LIN {X 0,Y 318.182,Z 547.875,A -85,B 0,C 180,E1 -15955.427,E2 -15955.427} C_VEL
LIN {X 0,Y 320.026,Z 530.036,A -85,B 0,C 180,E1 -15956.582,E2 -15956.582} C_VEL
LIN {X 0,Y 321.174,Z 516.208,A -85,B 0,C 180,E1 -15957.226,E2 -15957.226} C_VEL
LIN {X 0,Y 322.105,Z 502.779,A -85,B 0,C 180,E1 -15957.713,E2 -15957.713} C_VEL
LIN {X 0,Y 330.031,Z 435.019,A -85,B 0,C 180,E1 -15960.427,E2 -15960.427} C_VEL
LIN {X 0,Y 332.161,Z 417.671,A -85,B 0,C 180,E1 -15961.143,E2 -15961.143} C_VEL
LIN {X 0,Y 332.144,Z 415.549,A -85,B 0,C 180,E1 -15961.342,E2 -15961.342} C_VEL
LIN {X 0,Y 332.385,Z 414.109,A -85,B 0,C 180,E1 -15961.515,E2 -15961.515} C_VEL
LIN {X 0,Y 332.046,Z 411.059,A -85,B 0,C 180,E1 -15962.153,E2 -15962.153} C_VEL
LIN {X 0,Y 331.408,Z 405.664,A -85,B 0,C 180,E1 -15963.462,E2 -15963.462} C_VEL
LIN {X 0,Y 330.123,Z 402.878,A -85,B 0,C 180,E1 -15964.617,E2 -15964.617} C_VEL
LIN {X 0,Y 327.789,Z 399.05,A -85,B 0,C 180,E1 -15966.896,E2 -15966.896} C_VEL
LIN {X 0,Y 326.226,Z 396.525,A -85,B 0,C 180,E1 -15969.144,E2 -15969.144} C_VEL
LIN {X 0,Y 325.461,Z 395.342,A -85,B 0,C 180,E1 -15970.906,E2 -15970.906} C_VEL
LIN {X 0,Y 324.942,Z 395.007,A -85,B 0,C 180,E1 -15972.662,E2 -15972.662} C_VEL
LIN {X 0,Y 324.638,Z 395.462,A -85,B 0,C 180,E1 -15974.405,E2 -15974.405} C_VEL
LIN {X 0,Y 324.653,Z 396.483,A -85,B 0,C 180,E1 -15976.154,E2 -15976.154} C_VEL
LIN {X 0,Y 324.963,Z 398.076,A -85,B 0,C 180,E1 -15977.899,E2 -15977.899} C_VEL
LIN {X 0,Y 325.669,Z 401.15,A -85,B 0,C 180,E1 -15980.222,E2 -15980.222} C_VEL
LIN {X 0,Y 326.682,Z 406.362,A -85,B 0,C 180,E1 -15982.96,E2 -15982.96} C_VEL
LIN {X 0,Y 327.403,Z 411.448,A -85,B 0,C 180,E1 -15985.029,E2 -15985.029} C_VEL
LIN {X 0,Y 327.833,Z 416.51,A -85,B 0,C 180,E1 -15986.73,E2 -15986.73} C_VEL
LIN {X 0,Y 327.465,Z 419.21,A -85,B 0,C 180,E1 -15987.399,E2 -15987.399} C_VEL
LIN {X 0,Y 329.647,Z 433.874,A -85,B 0,C 180,E1 -15989.149,E2 -15989.149} C_VEL
LIN {X 0,Y 331.611,Z 449.295,A -85,B 0,C 180,E1 -15990.644,E2 -15990.644} C_VEL
LIN {X 0,Y 332.453,Z 459.55,A -85,B 0,C 180,E1 -15991.459,E2 -15991.459} C_VEL
LIN {X 0,Y 324.883,Z 534.704,A -85,B 0,C 180,E1 -15994.364,E2 -15994.364} C_VEL
LIN {X 0,Y 322.805,Z 549.723,A -85,B 0,C 180,E1 -15995.222,E2 -15995.222} C_VEL
LIN {X 0,Y 320.608,Z 562.727,A -85,B 0,C 180,E1 -15996.247,E2 -15996.247} C_VEL
LIN {X 0,Y 318.379,Z 574.516,A -85,B 0,C 180,E1 -15997.447,E2 -15997.447} C_VEL
LIN {X 0,Y 315.803,Z 586.406,A -85,B 0,C 180,E1 -15998.97,E2 -15998.97} C_VEL
LIN {X 0,Y 313.366,Z 596.431,A -85,B 0,C 180,E1 -16000.571,E2 -16000.571} C_VEL
LIN {X 0,Y 311.237,Z 604.933,A -85,B 0,C 180,E1 -16002.251,E2 -16002.251} C_VEL
LIN {X 0,Y 309.091,Z 612.857,A -85,B 0,C 180,E1 -16004.166,E2 -16004.166} C_VEL
LIN {X 0,Y 307.572,Z 619.204,A -85,B 0,C 180,E1 -16006.118,E2 -16006.118} C_VEL
LIN {X 0,Y 306.235,Z 624.295,A -85,B 0,C 180,E1 -16008.08,E2 -16008.08} C_VEL
LIN {X 0,Y 305.158,Z 628.243,A -85,B 0,C 180,E1 -16010.054,E2 -16010.054} C_VEL
LIN {X 0,Y 304.385,Z 631.13,A -85,B 0,C 180,E1 -16012.037,E2 -16012.037} C_VEL
LIN {X 0,Y 303.995,Z 632.859,A -85,B 0,C 180,E1 -16013.787,E2 -16013.787} C_VEL
LIN {X 0,Y 303.692,Z 633.934,A -85,B 0,C 180,E1 -16016.019,E2 -16016.019} C_VEL
LIN {X 0,Y 303.606,Z 633.986,A -85,B 0,C 180,E1 -16017.347,E2 -16017.347} C_VEL
LIN {X 0,Y 303.535,Z 633.619,A -85,B 0,C 180,E1 -16018.673,E2 -16018.673} C_VEL
LIN {X 0,Y 303.515,Z 632.811,A -85,B 0,C 180,E1 -16020,E2 -16020} C_VEL
LIN {X 0,Y 303.532,Z 631.523,A -85,B 0,C 180,E1 -16021.327,E2 -16021.327} C_VEL
LIN {X 0,Y 303.667,Z 628.745,A -85,B 0,C 180,E1 -16023.317,E2 -16023.317} C_VEL
LIN {X 0,Y 303.691,Z 624.826,A -85,B 0,C 180,E1 -16025.311,E2 -16025.311} C_VEL
LIN {X 0,Y 303.942,Z 619.686,A -85,B 0,C 180,E1 -16027.307,E2 -16027.307} C_VEL
LIN {X 0,Y 304.298,Z 613.15,A -85,B 0,C 180,E1 -16029.304,E2 -16029.304} C_VEL
LIN {X 0,Y 304.814,Z 604.894,A -85,B 0,C 180,E1 -16031.302,E2 -16031.302} C_VEL
LIN {X 0,Y 305.528,Z 596.499,A -85,B 0,C 180,E1 -16032.961,E2 -16032.961} C_VEL
LIN {X 0,Y 306.26,Z 587.38,A -85,B 0,C 180,E1 -16034.451,E2 -16034.451} C_VEL
LIN {X 0,Y 307.145,Z 576.203,A -85,B 0,C 180,E1 -16035.937,E2 -16035.937} C_VEL
LIN {X 0,Y 308.041,Z 563.777,A -85,B 0,C 180,E1 -16037.253,E2 -16037.253} C_VEL
LIN {X 0,Y 308.857,Z 550.689,A -85,B 0,C 180,E1 -16038.319,E2 -16038.319} C_VEL
LIN {X 0,Y 309.631,Z 537.051,A -85,B 0,C 180,E1 -16039.129,E2 -16039.129} C_VEL
LIN {X 0,Y 310.165,Z 522.846,A -85,B 0,C 180,E1 -16039.697,E2 -16039.697} C_VEL
LIN {X 0,Y 312.404,Z 451.025,A -85,B 0,C 180,E1 -16042.076,E2 -16042.076} C_VEL
LIN {X 0,Y 309.46,Z 422.574,A -85,B 0,C 180,E1 -16043.175,E2 -16043.175} C_VEL
LIN {X 0,Y 309.339,Z 419.877,A -85,B 0,C 180,E1 -16043.339,E2 -16043.339} C_VEL
LIN {X 0,Y 310.896,Z 400.877,A -85,B 0,C 180,E1 -16046.879,E2 -16046.879} C_VEL
LIN {X 0,Y 311.786,Z 389.598,A -85,B 0,C 180,E1 -16048.988,E2 -16048.988} C_VEL
LIN {X 0,Y 308.814,Z 375.793,A -85,B 0,C 180,E1 -16051.827,E2 -16051.827} C_VEL
LIN {X 0,Y 305.536,Z 361.201,A -85,B 0,C 180,E1 -16054.969,E2 -16054.969} C_VEL
LIN {X 0,Y 305.455,Z 361.063,A -85,B 0,C 180,E1 -16058.528,E2 -16058.528} C_VEL
LIN {X 0,Y 305.461,Z 361.055,A -85,B 0,C 180,E1 -16062.585,E2 -16062.585} C_VEL
LIN {X 0,Y 305.431,Z 361.045,A -85,B 0,C 180,E1 -16066.344,E2 -16066.344} C_VEL
LIN {X 0,Y 305.464,Z 361.04,A -85,B 0,C 180,E1 -16069.892,E2 -16069.892} C_VEL
LIN {X 0,Y 305.509,Z 361.129,A -85,B 0,C 180,E1 -16073.831,E2 -16073.831} C_VEL
LIN {X 0,Y 306.963,Z 366.882,A -85,B 0,C 180,E1 -16075.879,E2 -16075.879} C_VEL
LIN {X 0,Y 308.34,Z 372.284,A -85,B 0,C 180,E1 -16077.59,E2 -16077.59} C_VEL
LIN {X 0,Y 316.163,Z 388.914,A -85,B 0,C 180,E1 -16078.96,E2 -16078.96} C_VEL
LIN {X 0,Y 322.479,Z 404.145,A -85,B 0,C 180,E1 -16080.018,E2 -16080.018} C_VEL
LIN {X 0,Y 324.452,Z 415.875,A -85,B 0,C 180,E1 -16080.511,E2 -16080.511} C_VEL
LIN {X 0,Y 321.971,Z 498.445,A -85,B 0,C 180,E1 -16082.319,E2 -16082.319} C_VEL
LIN {X 0,Y 321.342,Z 514.068,A -85,B 0,C 180,E1 -16082.746,E2 -16082.746} C_VEL
LIN {X 0,Y 320.191,Z 527.937,A -85,B 0,C 180,E1 -16083.345,E2 -16083.345} C_VEL
LIN {X 0,Y 318.78,Z 541.464,A -85,B 0,C 180,E1 -16084.187,E2 -16084.187} C_VEL
LIN {X 0,Y 317.108,Z 554.588,A -85,B 0,C 180,E1 -16085.277,E2 -16085.277} C_VEL
LIN {X 0,Y 315.332,Z 566.41,A -85,B 0,C 180,E1 -16086.521,E2 -16086.521} C_VEL
LIN {X 0,Y 313.251,Z 578.455,A -85,B 0,C 180,E1 -16088.098,E2 -16088.098} C_VEL
LIN {X 0,Y 311.184,Z 589.311,A -85,B 0,C 180,E1 -16089.852,E2 -16089.852} C_VEL
LIN {X 0,Y 309.222,Z 599.086,A -85,B 0,C 180,E1 -16091.788,E2 -16091.788} C_VEL
LIN {X 0,Y 307.761,Z 606.494,A -85,B 0,C 180,E1 -16093.559,E2 -16093.559} C_VEL
LIN {X 0,Y 306.497,Z 613.955,A -85,B 0,C 180,E1 -16095.728,E2 -16095.728} C_VEL
LIN {X 0,Y 305.183,Z 620.391,A -85,B 0,C 180,E1 -16098.037,E2 -16098.037} C_VEL
LIN {X 0,Y 304.31,Z 626.095,A -85,B 0,C 180,E1 -16100.695,E2 -16100.695} C_VEL
LIN {X 0,Y 303.832,Z 630.239,A -85,B 0,C 180,E1 -16103.357,E2 -16103.357} C_VEL
LIN {X 0,Y 303.606,Z 632.954,A -85,B 0,C 180,E1 -16106.016,E2 -16106.016} C_VEL
LIN {X 0,Y 303.527,Z 634.316,A -85,B 0,C 180,E1 -16108.672,E2 -16108.672} C_VEL
LIN {X 0,Y 303.526,Z 634.349,A -85,B 0,C 180,E1 -16111.325,E2 -16111.325} C_VEL
LIN {X 0,Y 303.603,Z 633.053,A -85,B 0,C 180,E1 -16113.98,E2 -16113.98} C_VEL
LIN {X 0,Y 303.83,Z 630.396,A -85,B 0,C 180,E1 -16116.64,E2 -16116.64} C_VEL
LIN {X 0,Y 304.303,Z 626.307,A -85,B 0,C 180,E1 -16119.302,E2 -16119.302} C_VEL
LIN {X 0,Y 305.143,Z 620.663,A -85,B 0,C 180,E1 -16121.962,E2 -16121.962} C_VEL
LIN {X 0,Y 306.457,Z 614.298,A -85,B 0,C 180,E1 -16124.27,E2 -16124.27} C_VEL
LIN {X 0,Y 307.777,Z 606.859,A -85,B 0,C 180,E1 -16126.451,E2 -16126.451} C_VEL
LIN {X 0,Y 309.476,Z 598.103,A -85,B 0,C 180,E1 -16128.536,E2 -16128.536} C_VEL
LIN {X 0,Y 311.411,Z 588.131,A -85,B 0,C 180,E1 -16130.474,E2 -16130.474} C_VEL
LIN {X 0,Y 313.545,Z 577.03,A -85,B 0,C 180,E1 -16132.223,E2 -16132.223} C_VEL
LIN {X 0,Y 315.477,Z 565.984,A -85,B 0,C 180,E1 -16133.638,E2 -16133.638} C_VEL
LIN {X 0,Y 317.275,Z 553.988,A -85,B 0,C 180,E1 -16134.888,E2 -16134.888} C_VEL
LIN {X 0,Y 318.927,Z 540.711,A -85,B 0,C 180,E1 -16135.973,E2 -16135.973} C_VEL
LIN {X 0,Y 320.323,Z 526.914,A -85,B 0,C 180,E1 -16136.815,E2 -16136.815} C_VEL
LIN {X 0,Y 321.461,Z 512.549,A -85,B 0,C 180,E1 -16137.416,E2 -16137.416} C_VEL
LIN {X 0,Y 322.286,Z 492.491,A -85,B 0,C 180,E1 -16137.913,E2 -16137.913} C_VEL
LIN {X 0,Y 322.395,Z 488.057,A -85,B 0,C 180,E1 -16138.012,E2 -16138.012} C_VEL
LIN {X 0,Y 322.01,Z 482.254,A -85,B 0,C 180,E1 -16138.192,E2 -16138.192} C_VEL
LIN {X 0,Y 317.564,Z 463.594,A -85,B 0,C 180,E1 -16139.095,E2 -16139.095} C_VEL
LIN {X 0,Y 317.105,Z 457.794,A -85,B 0,C 180,E1 -16139.288,E2 -16139.288} C_VEL
LIN {X 0,Y 318.252,Z 415.603,A -85,B 0,C 180,E1 -16140.246,E2 -16140.246} C_VEL
LIN {X 0,Y 316.291,Z 405.8,A -85,B 0,C 180,E1 -16140.706,E2 -16140.706} C_VEL
LIN {X 0,Y 309.273,Z 389.276,A -85,B 0,C 180,E1 -16141.923,E2 -16141.923} C_VEL
LIN {X 0,Y 301.176,Z 372.441,A -85,B 0,C 180,E1 -16143.389,E2 -16143.389} C_VEL
LIN {X 0,Y 300.133,Z 368.625,A -85,B 0,C 180,E1 -16144.591,E2 -16144.591} C_VEL
LIN {X 0,Y 298.468,Z 361.978,A -85,B 0,C 180,E1 -16147.021,E2 -16147.021} C_VEL
LIN {X 0,Y 298.451,Z 361.921,A -85,B 0,C 180,E1 -16151.248,E2 -16151.248} C_VEL
LIN {X 0,Y 298.483,Z 361.897,A -85,B 0,C 180,E1 -16155.059,E2 -16155.059} C_VEL
LIN {X 0,Y 298.452,Z 361.934,A -85,B 0,C 180,E1 -16158.895,E2 -16158.895} C_VEL
LIN {X 0,Y 298.458,Z 361.893,A -85,B 0,C 180,E1 -16163.186,E2 -16163.186} C_VEL
LIN {X 0,Y 298.388,Z 361.939,A -85,B 0,C 180,E1 -16167.199,E2 -16167.199} C_VEL
LIN {X 0,Y 298.423,Z 361.878,A -85,B 0,C 180,E1 -16170.614,E2 -16170.614} C_VEL
LIN {X 0,Y 298.475,Z 361.904,A -85,B 0,C 180,E1 -16173.473,E2 -16173.473} C_VEL
LIN {X 0,Y 298.427,Z 361.936,A -85,B 0,C 180,E1 -16176.696,E2 -16176.696} C_VEL
LIN {X 0,Y 298.53,Z 361.919,A -85,B 0,C 180,E1 -16180.756,E2 -16180.756} C_VEL
LIN {X 0,Y 298.583,Z 361.897,A -85,B 0,C 180,E1 -16184.994,E2 -16184.994} C_VEL
LIN {X 0,Y 298.585,Z 361.902,A -85,B 0,C 180,E1 -16189.146,E2 -16189.146} C_VEL
LIN {X 0,Y 298.748,Z 361.884,A -85,B 0,C 180,E1 -16191.886,E2 -16191.886} C_VEL
LIN {X 0,Y 298.652,Z 361.905,A -85,B 0,C 180,E1 -16194.599,E2 -16194.599} C_VEL
LIN {X 0,Y 298.917,Z 361.868,A -85,B 0,C 180,E1 -16198.653,E2 -16198.653} C_VEL
LIN {X 0,Y 299.034,Z 361.86,A -85,B 0,C 180,E1 -16200,E2 -16200} C_VEL
LIN {X 0,Y 298.828,Z 361.868,A -85,B 0,C 180,E1 -16202.696,E2 -16202.696} C_VEL
LIN {X 0,Y 298.788,Z 361.891,A -85,B 0,C 180,E1 -16206.754,E2 -16206.754} C_VEL
LIN {X 0,Y 298.67,Z 361.883,A -85,B 0,C 180,E1 -16209.481,E2 -16209.481} C_VEL
LIN {X 0,Y 298.543,Z 361.914,A -85,B 0,C 180,E1 -16213.616,E2 -16213.616} C_VEL
LIN {X 0,Y 298.538,Z 361.903,A -85,B 0,C 180,E1 -16216.409,E2 -16216.409} C_VEL
LIN {X 0,Y 298.502,Z 361.92,A -85,B 0,C 180,E1 -16219.656,E2 -16219.656} C_VEL
LIN {X 0,Y 298.448,Z 361.932,A -85,B 0,C 180,E1 -16223.598,E2 -16223.598} C_VEL
LIN {X 0,Y 298.473,Z 361.904,A -85,B 0,C 180,E1 -16226.576,E2 -16226.576} C_VEL
LIN {X 0,Y 298.394,Z 361.882,A -85,B 0,C 180,E1 -16229.644,E2 -16229.644} C_VEL
LIN {X 0,Y 298.384,Z 361.938,A -85,B 0,C 180,E1 -16232.802,E2 -16232.802} C_VEL
LIN {X 0,Y 298.457,Z 361.893,A -85,B 0,C 180,E1 -16236.814,E2 -16236.814} C_VEL
LIN {X 0,Y 298.452,Z 361.934,A -85,B 0,C 180,E1 -16241.25,E2 -16241.25} C_VEL
LIN {X 0,Y 298.482,Z 361.897,A -85,B 0,C 180,E1 -16245.062,E2 -16245.062} C_VEL
LIN {X 0,Y 298.45,Z 361.92,A -85,B 0,C 180,E1 -16248.898,E2 -16248.898} C_VEL
LIN {X 0,Y 298.468,Z 362.013,A -85,B 0,C 180,E1 -16253.044,E2 -16253.044} C_VEL
LIN {X 0,Y 300.449,Z 369.766,A -85,B 0,C 180,E1 -16255.85,E2 -16255.85} C_VEL
LIN {X 0,Y 301.11,Z 372.24,A -85,B 0,C 180,E1 -16256.627,E2 -16256.627} C_VEL
LIN {X 0,Y 308.478,Z 387.538,A -85,B 0,C 180,E1 -16257.984,E2 -16257.984} C_VEL
LIN {X 0,Y 316.033,Z 405.034,A -85,B 0,C 180,E1 -16259.291,E2 -16259.291} C_VEL
LIN {X 0,Y 317.506,Z 411.383,A -85,B 0,C 180,E1 -16259.612,E2 -16259.612} C_VEL
LIN {X 0,Y 318.332,Z 416.622,A -85,B 0,C 180,E1 -16259.833,E2 -16259.833} C_VEL
LIN {X 0,Y 315.898,Z 494.268,A -85,B 0,C 180,E1 -16261.562,E2 -16261.562} C_VEL
LIN {X 0,Y 315.218,Z 512.539,A -85,B 0,C 180,E1 -16262.039,E2 -16262.039} C_VEL
LIN {X 0,Y 314.041,Z 526.906,A -85,B 0,C 180,E1 -16262.649,E2 -16262.649} C_VEL
LIN {X 0,Y 312.551,Z 540.139,A -85,B 0,C 180,E1 -16263.457,E2 -16263.457} C_VEL
LIN {X 0,Y 310.881,Z 553.549,A -85,B 0,C 180,E1 -16264.565,E2 -16264.565} C_VEL
LIN {X 0,Y 309.072,Z 565.636,A -85,B 0,C 180,E1 -16265.841,E2 -16265.841} C_VEL
LIN {X 0,Y 306.791,Z 577.83,A -85,B 0,C 180,E1 -16267.438,E2 -16267.438} C_VEL
LIN {X 0,Y 304.814,Z 587.901,A -85,B 0,C 180,E1 -16269.063,E2 -16269.063} C_VEL
LIN {X 0,Y 302.738,Z 597.911,A -85,B 0,C 180,E1 -16271.036,E2 -16271.036} C_VEL
LIN {X 0,Y 300.823,Z 607.229,A -85,B 0,C 180,E1 -16273.308,E2 -16273.308} C_VEL
LIN {X 0,Y 299.357,Z 615.173,A -85,B 0,C 180,E1 -16275.731,E2 -16275.731} C_VEL
LIN {X 0,Y 298.172,Z 620.557,A -85,B 0,C 180,E1 -16277.755,E2 -16277.755} C_VEL
LIN {X 0,Y 297.268,Z 626.225,A -85,B 0,C 180,E1 -16280.476,E2 -16280.476} C_VEL
LIN {X 0,Y 296.745,Z 630.336,A -85,B 0,C 180,E1 -16283.201,E2 -16283.201} C_VEL
LIN {X 0,Y 296.511,Z 633.016,A -85,B 0,C 180,E1 -16285.924,E2 -16285.924} C_VEL
LIN {X 0,Y 296.447,Z 634.338,A -85,B 0,C 180,E1 -16288.643,E2 -16288.643} C_VEL
LIN {X 0,Y 296.448,Z 634.33,A -85,B 0,C 180,E1 -16291.36,E2 -16291.36} C_VEL
LIN {X 0,Y 296.625,Z 632.445,A -85,B 0,C 180,E1 -16295.666,E2 -16295.666} C_VEL
LIN {X 0,Y 296.843,Z 631.726,A -85,B 0,C 180,E1 -16296.8,E2 -16296.8} C_VEL
LIN {X 0,Y 297.059,Z 630.455,A -85,B 0,C 180,E1 -16298.162,E2 -16298.162} C_VEL
LIN {X 0,Y 297.678,Z 627.768,A -85,B 0,C 180,E1 -16300.201,E2 -16300.201} C_VEL
LIN {X 0,Y 298.488,Z 624.041,A -85,B 0,C 180,E1 -16302.236,E2 -16302.236} C_VEL
LIN {X 0,Y 299.721,Z 619.19,A -85,B 0,C 180,E1 -16304.255,E2 -16304.255} C_VEL
LIN {X 0,Y 301.314,Z 612.169,A -85,B 0,C 180,E1 -16306.556,E2 -16306.556} C_VEL
LIN {X 0,Y 303.075,Z 604.298,A -85,B 0,C 180,E1 -16308.595,E2 -16308.595} C_VEL
LIN {X 0,Y 305.146,Z 594.851,A -85,B 0,C 180,E1 -16310.564,E2 -16310.564} C_VEL
LIN {X 0,Y 307.109,Z 585.333,A -85,B 0,C 180,E1 -16312.186,E2 -16312.186} C_VEL
LIN {X 0,Y 309.295,Z 573.702,A -85,B 0,C 180,E1 -16313.788,E2 -16313.788} C_VEL
LIN {X 0,Y 311.179,Z 561.561,A -85,B 0,C 180,E1 -16315.16,E2 -16315.16} C_VEL
LIN {X 0,Y 312.961,Z 548.604,A -85,B 0,C 180,E1 -16316.294,E2 -16316.294} C_VEL
LIN {X 0,Y 314.492,Z 534.098,A -85,B 0,C 180,E1 -16317.267,E2 -16317.267} C_VEL
LIN {X 0,Y 316.409,Z 512.855,A -85,B 0,C 180,E1 -16318.256,E2 -16318.256} C_VEL
LIN {X 0,Y 328.061,Z 420.09,A -85,B 0,C 180,E1 -16322.059,E2 -16322.059} C_VEL
LIN {X 0,Y 327.883,Z 417.132,A -85,B 0,C 180,E1 -16322.362,E2 -16322.362} C_VEL
LIN {X 0,Y 327.312,Z 413.657,A -85,B 0,C 180,E1 -16323.133,E2 -16323.133} C_VEL
LIN {X 0,Y 326.869,Z 410.419,A -85,B 0,C 180,E1 -16323.99,E2 -16323.99} C_VEL
LIN {X 0,Y 324.961,Z 406.805,A -85,B 0,C 180,E1 -16325.729,E2 -16325.729} C_VEL
LIN {X 0,Y 322.672,Z 403.199,A -85,B 0,C 180,E1 -16328.362,E2 -16328.362} C_VEL
LIN {X 0,Y 321.345,Z 401.123,A -85,B 0,C 180,E1 -16331.006,E2 -16331.006} C_VEL
LIN {X 0,Y 320.772,Z 400.777,A -85,B 0,C 180,E1 -16332.783,E2 -16332.783} C_VEL
LIN {X 0,Y 320.308,Z 401.68,A -85,B 0,C 180,E1 -16335.402,E2 -16335.402} C_VEL
LIN {X 0,Y 320.558,Z 404.041,A -85,B 0,C 180,E1 -16338.197,E2 -16338.197} C_VEL
LIN {X 0,Y 321.17,Z 407.324,A -85,B 0,C 180,E1 -16340.61,E2 -16340.61} C_VEL
LIN {X 0,Y 321.833,Z 411.838,A -85,B 0,C 180,E1 -16342.963,E2 -16342.963} C_VEL
LIN {X 0,Y 322.325,Z 416.005,A -85,B 0,C 180,E1 -16344.7,E2 -16344.7} C_VEL
LIN {X 0,Y 322.667,Z 419.697,A -85,B 0,C 180,E1 -16345.94,E2 -16345.94} C_VEL
LIN {X 0,Y 323.66,Z 423.168,A -85,B 0,C 180,E1 -16346.604,E2 -16346.604} C_VEL
LIN {X 0,Y 325.648,Z 437.927,A -85,B 0,C 180,E1 -16348.394,E2 -16348.394} C_VEL
LIN {X 0,Y 327.174,Z 452.09,A -85,B 0,C 180,E1 -16349.814,E2 -16349.814} C_VEL
LIN {X 0,Y 327.787,Z 460.947,A -85,B 0,C 180,E1 -16350.55,E2 -16350.55} C_VEL
LIN {X 0,Y 319.743,Z 534.694,A -85,B 0,C 180,E1 -16353.482,E2 -16353.482} C_VEL
LIN {X 0,Y 317.564,Z 549.543,A -85,B 0,C 180,E1 -16354.346,E2 -16354.346} C_VEL
LIN {X 0,Y 315.066,Z 563.279,A -85,B 0,C 180,E1 -16355.452,E2 -16355.452} C_VEL
LIN {X 0,Y 312.672,Z 574.881,A -85,B 0,C 180,E1 -16356.662,E2 -16356.662} C_VEL
LIN {X 0,Y 309.938,Z 586.634,A -85,B 0,C 180,E1 -16358.204,E2 -16358.204} C_VEL
LIN {X 0,Y 307.202,Z 597.114,A -85,B 0,C 180,E1 -16359.93,E2 -16359.93} C_VEL
LIN {X 0,Y 304.647,Z 606.45,A -85,B 0,C 180,E1 -16361.854,E2 -16361.854} C_VEL
LIN {X 0,Y 302.36,Z 614.023,A -85,B 0,C 180,E1 -16363.804,E2 -16363.804} C_VEL
LIN {X 0,Y 300.743,Z 620.12,A -85,B 0,C 180,E1 -16365.796,E2 -16365.796} C_VEL
LIN {X 0,Y 299.343,Z 625,A -85,B 0,C 180,E1 -16367.801,E2 -16367.801} C_VEL
LIN {X 0,Y 298.188,Z 628.763,A -85,B 0,C 180,E1 -16369.819,E2 -16369.819} C_VEL
LIN {X 0,Y 297.374,Z 631.476,A -85,B 0,C 180,E1 -16371.848,E2 -16371.848} C_VEL
LIN {X 0,Y 296.88,Z 633.192,A -85,B 0,C 180,E1 -16373.869,E2 -16373.869} C_VEL
LIN {X 0,Y 296.598,Z 633.959,A -85,B 0,C 180,E1 -16375.924,E2 -16375.924} C_VEL
LIN {X 0,Y 296.514,Z 633.931,A -85,B 0,C 180,E1 -16377.283,E2 -16377.283} C_VEL
LIN {X 0,Y 296.457,Z 633.467,A -85,B 0,C 180,E1 -16378.642,E2 -16378.642} C_VEL
LIN {X 0,Y 296.434,Z 632.529,A -85,B 0,C 180,E1 -16380,E2 -16380} C_VEL
LIN {X 0,Y 296.454,Z 631.163,A -85,B 0,C 180,E1 -16381.359,E2 -16381.359} C_VEL
LIN {X 0,Y 296.602,Z 628.229,A -85,B 0,C 180,E1 -16383.396,E2 -16383.396} C_VEL
LIN {X 0,Y 296.672,Z 623.427,A -85,B 0,C 180,E1 -16385.744,E2 -16385.744} C_VEL
LIN {X 0,Y 296.937,Z 617.765,A -85,B 0,C 180,E1 -16387.822,E2 -16387.822} C_VEL
LIN {X 0,Y 297.319,Z 610.722,A -85,B 0,C 180,E1 -16389.868,E2 -16389.868} C_VEL
LIN {X 0,Y 297.826,Z 603.52,A -85,B 0,C 180,E1 -16391.571,E2 -16391.571} C_VEL
LIN {X 0,Y 298.566,Z 594.808,A -85,B 0,C 180,E1 -16393.268,E2 -16393.268} C_VEL
LIN {X 0,Y 299.482,Z 584.188,A -85,B 0,C 180,E1 -16394.96,E2 -16394.96} C_VEL
LIN {X 0,Y 300.336,Z 572.527,A -85,B 0,C 180,E1 -16396.45,E2 -16396.45} C_VEL
LIN {X 0,Y 301.219,Z 560.631,A -85,B 0,C 180,E1 -16397.657,E2 -16397.657} C_VEL
LIN {X 0,Y 302.001,Z 547.74,A -85,B 0,C 180,E1 -16398.662,E2 -16398.662} C_VEL
LIN {X 0,Y 302.784,Z 533.872,A -85,B 0,C 180,E1 -16399.447,E2 -16399.447} C_VEL
LIN {X 0,Y 303.969,Z 496.409,A -85,B 0,C 180,E1 -16400.779,E2 -16400.779} C_VEL
LIN {X 0,Y 305.461,Z 451.797,A -85,B 0,C 180,E1 -16402.315,E2 -16402.315} C_VEL
LIN {X 0,Y 302.673,Z 424.414,A -85,B 0,C 180,E1 -16403.408,E2 -16403.408} C_VEL
LIN {X 0,Y 302.372,Z 419.92,A -85,B 0,C 180,E1 -16403.637,E2 -16403.637} C_VEL
LIN {X 0,Y 303.973,Z 401.207,A -85,B 0,C 180,E1 -16407.17,E2 -16407.17} C_VEL
LIN {X 0,Y 304.856,Z 391.76,A -85,B 0,C 180,E1 -16408.955,E2 -16408.955} C_VEL
LIN {X 0,Y 304.253,Z 387.742,A -85,B 0,C 180,E1 -16409.778,E2 -16409.778} C_VEL
LIN {X 0,Y 300.433,Z 370.668,A -85,B 0,C 180,E1 -16413.395,E2 -16413.395} C_VEL
LIN {X 0,Y 298.489,Z 362.13,A -85,B 0,C 180,E1 -16415.278,E2 -16415.278} C_VEL
LIN {X 0,Y 298.41,Z 361.939,A -85,B 0,C 180,E1 -16418.993,E2 -16418.993} C_VEL
LIN {X 0,Y 298.405,Z 361.925,A -85,B 0,C 180,E1 -16423.103,E2 -16423.103} C_VEL
LIN {X 0,Y 298.409,Z 361.93,A -85,B 0,C 180,E1 -16426.92,E2 -16426.92} C_VEL
LIN {X 0,Y 298.421,Z 361.919,A -85,B 0,C 180,E1 -16431.003,E2 -16431.003} C_VEL
LIN {X 0,Y 298.467,Z 362.086,A -85,B 0,C 180,E1 -16433.187,E2 -16433.187} C_VEL
LIN {X 0,Y 300.828,Z 371.239,A -85,B 0,C 180,E1 -16436.428,E2 -16436.428} C_VEL
LIN {X 0,Y 301.24,Z 372.666,A -85,B 0,C 180,E1 -16436.763,E2 -16436.763} C_VEL
LIN {X 0,Y 310.282,Z 391.494,A -85,B 0,C 180,E1 -16438.372,E2 -16438.372} C_VEL
LIN {X 0,Y 316.529,Z 406.423,A -85,B 0,C 180,E1 -16439.453,E2 -16439.453} C_VEL
LIN {X 0,Y 318.269,Z 416.961,A -85,B 0,C 180,E1 -16439.907,E2 -16439.907} C_VEL
LIN {X 0,Y 315.704,Z 498.47,A -85,B 0,C 180,E1 -16441.72,E2 -16441.72} C_VEL
LIN {X 0,Y 315.059,Z 514.083,A -85,B 0,C 180,E1 -16442.155,E2 -16442.155} C_VEL
LIN {X 0,Y 313.879,Z 527.947,A -85,B 0,C 180,E1 -16442.765,E2 -16442.765} C_VEL
LIN {X 0,Y 312.409,Z 541.471,A -85,B 0,C 180,E1 -16443.62,E2 -16443.62} C_VEL
LIN {X 0,Y 310.609,Z 554.993,A -85,B 0,C 180,E1 -16444.769,E2 -16444.769} C_VEL
LIN {X 0,Y 308.823,Z 566.414,A -85,B 0,C 180,E1 -16445.995,E2 -16445.995} C_VEL
LIN {X 0,Y 306.654,Z 578.459,A -85,B 0,C 180,E1 -16447.602,E2 -16447.602} C_VEL
LIN {X 0,Y 304.484,Z 589.314,A -85,B 0,C 180,E1 -16449.389,E2 -16449.389} C_VEL
LIN {X 0,Y 302.463,Z 599.089,A -85,B 0,C 180,E1 -16451.366,E2 -16451.366} C_VEL
LIN {X 0,Y 300.818,Z 607.002,A -85,B 0,C 180,E1 -16453.312,E2 -16453.312} C_VEL
LIN {X 0,Y 299.365,Z 614.964,A -85,B 0,C 180,E1 -16455.728,E2 -16455.728} C_VEL
LIN {X 0,Y 298.198,Z 620.392,A -85,B 0,C 180,E1 -16457.752,E2 -16457.752} C_VEL
LIN {X 0,Y 297.275,Z 626.096,A -85,B 0,C 180,E1 -16460.473,E2 -16460.473} C_VEL
LIN {X 0,Y 296.747,Z 630.24,A -85,B 0,C 180,E1 -16463.198,E2 -16463.198} C_VEL
LIN {X 0,Y 296.51,Z 632.955,A -85,B 0,C 180,E1 -16465.921,E2 -16465.921} C_VEL
LIN {X 0,Y 296.449,Z 634.316,A -85,B 0,C 180,E1 -16468.64,E2 -16468.64} C_VEL
LIN {X 0,Y 296.448,Z 634.349,A -85,B 0,C 180,E1 -16471.357,E2 -16471.357} C_VEL
LIN {X 0,Y 296.507,Z 633.052,A -85,B 0,C 180,E1 -16474.076,E2 -16474.076} C_VEL
LIN {X 0,Y 296.746,Z 630.395,A -85,B 0,C 180,E1 -16476.799,E2 -16476.799} C_VEL
LIN {X 0,Y 297.267,Z 626.306,A -85,B 0,C 180,E1 -16479.524,E2 -16479.524} C_VEL
LIN {X 0,Y 298.16,Z 620.662,A -85,B 0,C 180,E1 -16482.246,E2 -16482.246} C_VEL
LIN {X 0,Y 299.551,Z 614.296,A -85,B 0,C 180,E1 -16484.607,E2 -16484.607} C_VEL
LIN {X 0,Y 301.046,Z 606.227,A -85,B 0,C 180,E1 -16487.008,E2 -16487.008} C_VEL
LIN {X 0,Y 302.716,Z 598.101,A -85,B 0,C 180,E1 -16488.965,E2 -16488.965} C_VEL
LIN {X 0,Y 304.757,Z 588.128,A -85,B 0,C 180,E1 -16490.941,E2 -16490.941} C_VEL
LIN {X 0,Y 306.941,Z 577.026,A -85,B 0,C 180,E1 -16492.728,E2 -16492.728} C_VEL
LIN {X 0,Y 309.131,Z 564.977,A -85,B 0,C 180,E1 -16494.282,E2 -16494.282} C_VEL
LIN {X 0,Y 311.074,Z 552.225,A -85,B 0,C 180,E1 -16495.598,E2 -16495.598} C_VEL
LIN {X 0,Y 312.767,Z 538.444,A -85,B 0,C 180,E1 -16496.704,E2 -16496.704} C_VEL
LIN {X 0,Y 314.241,Z 524.619,A -85,B 0,C 180,E1 -16497.513,E2 -16497.513} C_VEL
LIN {X 0,Y 315.242,Z 511.395,A -85,B 0,C 180,E1 -16498.049,E2 -16498.049} C_VEL
LIN {X 0,Y 316.155,Z 488.278,A -85,B 0,C 180,E1 -16498.609,E2 -16498.609} C_VEL
LIN {X 0,Y 317.105,Z 457.794,A -85,B 0,C 180,E1 -16499.288,E2 -16499.288} C_VEL
LIN {X 0,Y 316.648,Z 451.998,A -85,B 0,C 180,E1 -16499.482,E2 -16499.482} C_VEL
LIN {X 0,Y 312.255,Z 433.362,A -85,B 0,C 180,E1 -16500.424,E2 -16500.424} C_VEL
LIN {X 0,Y 311.861,Z 427.564,A -85,B 0,C 180,E1 -16500.619,E2 -16500.619} C_VEL
LIN {X 0,Y 312.098,Z 416.551,A -85,B 0,C 180,E1 -16500.882,E2 -16500.882} C_VEL
LIN {X 0,Y 310.358,Z 408.132,A -85,B 0,C 180,E1 -16501.297,E2 -16501.297} C_VEL
LIN {X 0,Y 302.987,Z 390.864,A -85,B 0,C 180,E1 -16502.622,E2 -16502.622} C_VEL
LIN {X 0,Y 295.244,Z 375.343,A -85,B 0,C 180,E1 -16504.033,E2 -16504.033} C_VEL
LIN {X 0,Y 293.745,Z 372.005,A -85,B 0,C 180,E1 -16504.409,E2 -16504.409} C_VEL
LIN {X 0,Y 291.435,Z 363.021,A -85,B 0,C 180,E1 -16507.66,E2 -16507.66} C_VEL
LIN {X 0,Y 291.401,Z 362.792,A -85,B 0,C 180,E1 -16510.628,E2 -16510.628} C_VEL
LIN {X 0,Y 291.4,Z 362.782,A -85,B 0,C 180,E1 -16514.378,E2 -16514.378} C_VEL
LIN {X 0,Y 291.387,Z 362.815,A -85,B 0,C 180,E1 -16518.388,E2 -16518.388} C_VEL
LIN {X 0,Y 291.374,Z 362.775,A -85,B 0,C 180,E1 -16521.161,E2 -16521.161} C_VEL
LIN {X 0,Y 291.377,Z 362.798,A -85,B 0,C 180,E1 -16524.628,E2 -16524.628} C_VEL
LIN {X 0,Y 291.364,Z 362.803,A -85,B 0,C 180,E1 -16527.95,E2 -16527.95} C_VEL
LIN {X 0,Y 291.373,Z 362.754,A -85,B 0,C 180,E1 -16531.157,E2 -16531.157} C_VEL
LIN {X 0,Y 291.408,Z 362.796,A -85,B 0,C 180,E1 -16534.271,E2 -16534.271} C_VEL
LIN {X 0,Y 291.373,Z 362.807,A -85,B 0,C 180,E1 -16537.299,E2 -16537.299} C_VEL
LIN {X 0,Y 291.448,Z 362.8,A -85,B 0,C 180,E1 -16540.269,E2 -16540.269} C_VEL
LIN {X 0,Y 291.545,Z 362.772,A -85,B 0,C 180,E1 -16544.623,E2 -16544.623} C_VEL
LIN {X 0,Y 291.529,Z 362.784,A -85,B 0,C 180,E1 -16548.88,E2 -16548.88} C_VEL
LIN {X 0,Y 291.699,Z 362.759,A -85,B 0,C 180,E1 -16551.688,E2 -16551.688} C_VEL
LIN {X 0,Y 291.623,Z 362.782,A -85,B 0,C 180,E1 -16554.468,E2 -16554.468} C_VEL
LIN {X 0,Y 291.883,Z 362.744,A -85,B 0,C 180,E1 -16558.62,E2 -16558.62} C_VEL
LIN {X 0,Y 291.883,Z 362.745,A -85,B 0,C 180,E1 -16561.38,E2 -16561.38} C_VEL
LIN {X 0,Y 291.736,Z 362.768,A -85,B 0,C 180,E1 -16566.918,E2 -16566.918} C_VEL
LIN {X 0,Y 291.619,Z 362.76,A -85,B 0,C 180,E1 -16569.712,E2 -16569.712} C_VEL
LIN {X 0,Y 291.513,Z 362.788,A -85,B 0,C 180,E1 -16573.951,E2 -16573.951} C_VEL
LIN {X 0,Y 291.477,Z 362.786,A -85,B 0,C 180,E1 -16576.818,E2 -16576.818} C_VEL
LIN {X 0,Y 291.441,Z 362.797,A -85,B 0,C 180,E1 -16579.875,E2 -16579.875} C_VEL
LIN {X 0,Y 291.39,Z 362.814,A -85,B 0,C 180,E1 -16584.206,E2 -16584.206} C_VEL
LIN {X 0,Y 291.402,Z 362.766,A -85,B 0,C 180,E1 -16587.274,E2 -16587.274} C_VEL
LIN {X 0,Y 291.314,Z 362.772,A -85,B 0,C 180,E1 -16590.439,E2 -16590.439} C_VEL
LIN {X 0,Y 291.335,Z 362.821,A -85,B 0,C 180,E1 -16593.7,E2 -16593.7} C_VEL
LIN {X 0,Y 291.39,Z 362.768,A -85,B 0,C 180,E1 -16597.261,E2 -16597.261} C_VEL
LIN {X 0,Y 291.4,Z 362.804,A -85,B 0,C 180,E1 -16600.631,E2 -16600.631} C_VEL
LIN {X 0,Y 291.4,Z 362.779,A -85,B 0,C 180,E1 -16604.381,E2 -16604.381} C_VEL
LIN {X 0,Y 291.385,Z 362.807,A -85,B 0,C 180,E1 -16608.391,E2 -16608.391} C_VEL
LIN {X 0,Y 291.434,Z 362.956,A -85,B 0,C 180,E1 -16612.339,E2 -16612.339} C_VEL
LIN {X 0,Y 293.755,Z 371.971,A -85,B 0,C 180,E1 -16615.628,E2 -16615.628} C_VEL
LIN {X 0,Y 295.312,Z 375.394,A -85,B 0,C 180,E1 -16616.022,E2 -16616.022} C_VEL
LIN {X 0,Y 303.33,Z 391.645,A -85,B 0,C 180,E1 -16617.486,E2 -16617.486} C_VEL
LIN {X 0,Y 310.469,Z 408.407,A -85,B 0,C 180,E1 -16618.768,E2 -16618.768} C_VEL
LIN {X 0,Y 312.16,Z 416.779,A -85,B 0,C 180,E1 -16619.176,E2 -16619.176} C_VEL
LIN {X 0,Y 309.69,Z 494.289,A -85,B 0,C 180,E1 -16620.938,E2 -16620.938} C_VEL
LIN {X 0,Y 308.965,Z 512.553,A -85,B 0,C 180,E1 -16621.421,E2 -16621.421} C_VEL
LIN {X 0,Y 307.739,Z 526.915,A -85,B 0,C 180,E1 -16622.04,E2 -16622.04} C_VEL
LIN {X 0,Y 306.086,Z 541.275,A -85,B 0,C 180,E1 -16622.943,E2 -16622.943} C_VEL
LIN {X 0,Y 304.3,Z 554.723,A -85,B 0,C 180,E1 -16624.103,E2 -16624.103} C_VEL
LIN {X 0,Y 302.356,Z 566.953,A -85,B 0,C 180,E1 -16625.452,E2 -16625.452} C_VEL
LIN {X 0,Y 300.036,Z 578.902,A -85,B 0,C 180,E1 -16627.084,E2 -16627.084} C_VEL
LIN {X 0,Y 297.796,Z 589.685,A -85,B 0,C 180,E1 -16628.908,E2 -16628.908} C_VEL
LIN {X 0,Y 295.671,Z 599.398,A -85,B 0,C 180,E1 -16630.925,E2 -16630.925} C_VEL
LIN {X 0,Y 293.896,Z 607.716,A -85,B 0,C 180,E1 -16633.044,E2 -16633.044} C_VEL
LIN {X 0,Y 292.463,Z 615.174,A -85,B 0,C 180,E1 -16635.387,E2 -16635.387} C_VEL
LIN {X 0,Y 291.199,Z 620.558,A -85,B 0,C 180,E1 -16637.457,E2 -16637.457} C_VEL
LIN {X 0,Y 290.247,Z 626.226,A -85,B 0,C 180,E1 -16640.243,E2 -16640.243} C_VEL
LIN {X 0,Y 289.671,Z 630.337,A -85,B 0,C 180,E1 -16643.034,E2 -16643.034} C_VEL
LIN {X 0,Y 289.42,Z 633.016,A -85,B 0,C 180,E1 -16645.824,E2 -16645.824} C_VEL
LIN {X 0,Y 289.371,Z 634.338,A -85,B 0,C 180,E1 -16648.61,E2 -16648.61} C_VEL
LIN {X 0,Y 289.371,Z 634.33,A -85,B 0,C 180,E1 -16651.393,E2 -16651.393} C_VEL
LIN {X 0,Y 289.416,Z 633.007,A -85,B 0,C 180,E1 -16654.179,E2 -16654.179} C_VEL
LIN {X 0,Y 289.769,Z 631.982,A -85,B 0,C 180,E1 -16656.967,E2 -16656.967} C_VEL
LIN {X 0,Y 290.038,Z 630.864,A -85,B 0,C 180,E1 -16658.361,E2 -16658.361} C_VEL
LIN {X 0,Y 290.708,Z 628.344,A -85,B 0,C 180,E1 -16660.448,E2 -16660.448} C_VEL
LIN {X 0,Y 291.589,Z 624.839,A -85,B 0,C 180,E1 -16662.53,E2 -16662.53} C_VEL
LIN {X 0,Y 292.912,Z 620.209,A -85,B 0,C 180,E1 -16664.594,E2 -16664.594} C_VEL
LIN {X 0,Y 294.673,Z 613.317,A -85,B 0,C 180,E1 -16666.991,E2 -16666.991} C_VEL
LIN {X 0,Y 296.552,Z 605.942,A -85,B 0,C 180,E1 -16669.019,E2 -16669.019} C_VEL
LIN {X 0,Y 298.785,Z 596.955,A -85,B 0,C 180,E1 -16671.023,E2 -16671.023} C_VEL
LIN {X 0,Y 300.859,Z 587.876,A -85,B 0,C 180,E1 -16672.672,E2 -16672.672} C_VEL
LIN {X 0,Y 303.245,Z 577.018,A -85,B 0,C 180,E1 -16674.293,E2 -16674.293} C_VEL
LIN {X 0,Y 305.685,Z 563.593,A -85,B 0,C 180,E1 -16675.903,E2 -16675.903} C_VEL
LIN {X 0,Y 307.678,Z 550.912,A -85,B 0,C 180,E1 -16677.084,E2 -16677.084} C_VEL
LIN {X 0,Y 309.497,Z 536.502,A -85,B 0,C 180,E1 -16678.113,E2 -16678.113} C_VEL
LIN {X 0,Y 311.331,Z 518.148,A -85,B 0,C 180,E1 -16679.036,E2 -16679.036} C_VEL
LIN {X 0,Y 314.544,Z 492.304,A -85,B 0,C 180,E1 -16680.136,E2 -16680.136} C_VEL
LIN {X 0,Y 324.258,Z 421.932,A -85,B 0,C 180,E1 -16683.079,E2 -16683.079} C_VEL
LIN {X 0,Y 322.657,Z 416.472,A -85,B 0,C 180,E1 -16684.137,E2 -16684.137} C_VEL
LIN {X 0,Y 322.367,Z 415.216,A -85,B 0,C 180,E1 -16684.531,E2 -16684.531} C_VEL
LIN {X 0,Y 320.434,Z 411.863,A -85,B 0,C 180,E1 -16686.314,E2 -16686.314} C_VEL
LIN {X 0,Y 318.896,Z 409.42,A -85,B 0,C 180,E1 -16688.105,E2 -16688.105} C_VEL
LIN {X 0,Y 317.808,Z 407.652,A -85,B 0,C 180,E1 -16689.891,E2 -16689.891} C_VEL
LIN {X 0,Y 317.045,Z 406.69,A -85,B 0,C 180,E1 -16691.685,E2 -16691.685} C_VEL
LIN {X 0,Y 316.425,Z 406.649,A -85,B 0,C 180,E1 -16693.516,E2 -16693.516} C_VEL
LIN {X 0,Y 316.037,Z 408.038,A -85,B 0,C 180,E1 -16696.419,E2 -16696.419} C_VEL
LIN {X 0,Y 316.279,Z 410.675,A -85,B 0,C 180,E1 -16699.072,E2 -16699.072} C_VEL
LIN {X 0,Y 316.727,Z 414.65,A -85,B 0,C 180,E1 -16701.588,E2 -16701.588} C_VEL
LIN {X 0,Y 317.257,Z 419.16,A -85,B 0,C 180,E1 -16703.734,E2 -16703.734} C_VEL
LIN {X 0,Y 319.902,Z 426.204,A -85,B 0,C 180,E1 -16705.581,E2 -16705.581} C_VEL
LIN {X 0,Y 320.288,Z 428.783,A -85,B 0,C 180,E1 -16705.975,E2 -16705.975} C_VEL
LIN {X 0,Y 321.804,Z 442.222,A -85,B 0,C 180,E1 -16707.646,E2 -16707.646} C_VEL
LIN {X 0,Y 323,Z 456.301,A -85,B 0,C 180,E1 -16709.075,E2 -16709.075} C_VEL
LIN {X 0,Y 323.294,Z 462.639,A -85,B 0,C 180,E1 -16709.613,E2 -16709.613} C_VEL
LIN {X 0,Y 314.746,Z 535.193,A -85,B 0,C 180,E1 -16712.578,E2 -16712.578} C_VEL
LIN {X 0,Y 312.429,Z 549.736,A -85,B 0,C 180,E1 -16713.443,E2 -16713.443} C_VEL
LIN {X 0,Y 309.926,Z 562.487,A -85,B 0,C 180,E1 -16714.478,E2 -16714.478} C_VEL
LIN {X 0,Y 307.373,Z 574.182,A -85,B 0,C 180,E1 -16715.697,E2 -16715.697} C_VEL
LIN {X 0,Y 304.121,Z 587.05,A -85,B 0,C 180,E1 -16717.407,E2 -16717.407} C_VEL
LIN {X 0,Y 301.228,Z 597.371,A -85,B 0,C 180,E1 -16719.157,E2 -16719.157} C_VEL
LIN {X 0,Y 298.48,Z 606.622,A -85,B 0,C 180,E1 -16721.11,E2 -16721.11} C_VEL
LIN {X 0,Y 296.094,Z 614.113,A -85,B 0,C 180,E1 -16723.096,E2 -16723.096} C_VEL
LIN {X 0,Y 293.93,Z 621.098,A -85,B 0,C 180,E1 -16725.46,E2 -16725.46} C_VEL
LIN {X 0,Y 292.46,Z 625.748,A -85,B 0,C 180,E1 -16727.51,E2 -16727.51} C_VEL
LIN {X 0,Y 291.23,Z 629.313,A -85,B 0,C 180,E1 -16729.573,E2 -16729.573} C_VEL
LIN {X 0,Y 290.347,Z 631.846,A -85,B 0,C 180,E1 -16731.649,E2 -16731.649} C_VEL
LIN {X 0,Y 289.764,Z 633.51,A -85,B 0,C 180,E1 -16733.958,E2 -16733.958} C_VEL
LIN {X 0,Y 289.508,Z 633.985,A -85,B 0,C 180,E1 -16735.824,E2 -16735.824} C_VEL
LIN {X 0,Y 289.424,Z 633.85,A -85,B 0,C 180,E1 -16737.216,E2 -16737.216} C_VEL
LIN {X 0,Y 289.381,Z 633.25,A -85,B 0,C 180,E1 -16738.608,E2 -16738.608} C_VEL
LIN {X 0,Y 289.356,Z 632.231,A -85,B 0,C 180,E1 -16740,E2 -16740} C_VEL
LIN {X 0,Y 289.378,Z 630.771,A -85,B 0,C 180,E1 -16741.392,E2 -16741.392} C_VEL
LIN {X 0,Y 289.538,Z 627.669,A -85,B 0,C 180,E1 -16743.479,E2 -16743.479} C_VEL
LIN {X 0,Y 289.6,Z 623.008,A -85,B 0,C 180,E1 -16745.728,E2 -16745.728} C_VEL
LIN {X 0,Y 289.891,Z 616.766,A -85,B 0,C 180,E1 -16748.013,E2 -16748.013} C_VEL
LIN {X 0,Y 290.294,Z 609.459,A -85,B 0,C 180,E1 -16750.109,E2 -16750.109} C_VEL
LIN {X 0,Y 290.971,Z 600.333,A -85,B 0,C 180,E1 -16752.201,E2 -16752.201} C_VEL
LIN {X 0,Y 291.713,Z 590.955,A -85,B 0,C 180,E1 -16753.941,E2 -16753.941} C_VEL
LIN {X 0,Y 292.651,Z 579.939,A -85,B 0,C 180,E1 -16755.599,E2 -16755.599} C_VEL
LIN {X 0,Y 293.509,Z 569.469,A -85,B 0,C 180,E1 -16756.878,E2 -16756.878} C_VEL
LIN {X 0,Y 294.451,Z 556.028,A -85,B 0,C 180,E1 -16758.167,E2 -16758.167} C_VEL
LIN {X 0,Y 295.229,Z 543.017,A -85,B 0,C 180,E1 -16759.106,E2 -16759.106} C_VEL
LIN {X 0,Y 295.99,Z 528.964,A -85,B 0,C 180,E1 -16759.822,E2 -16759.822} C_VEL
LIN {X 0,Y 298.525,Z 452.43,A -85,B 0,C 180,E1 -16762.556,E2 -16762.556} C_VEL
LIN {X 0,Y 295.844,Z 426.587,A -85,B 0,C 180,E1 -16763.616,E2 -16763.616} C_VEL
LIN {X 0,Y 295.418,Z 420.153,A -85,B 0,C 180,E1 -16763.902,E2 -16763.902} C_VEL
LIN {X 0,Y 296.87,Z 403.384,A -85,B 0,C 180,E1 -16767.111,E2 -16767.111} C_VEL
LIN {X 0,Y 297.896,Z 392.547,A -85,B 0,C 180,E1 -16769.199,E2 -16769.199} C_VEL
LIN {X 0,Y 295.126,Z 379.359,A -85,B 0,C 180,E1 -16771.996,E2 -16771.996} C_VEL
LIN {X 0,Y 291.434,Z 362.981,A -85,B 0,C 180,E1 -16775.629,E2 -16775.629} C_VEL
LIN {X 0,Y 291.387,Z 362.814,A -85,B 0,C 180,E1 -16779.481,E2 -16779.481} C_VEL
LIN {X 0,Y 291.314,Z 362.798,A -85,B 0,C 180,E1 -16783.633,E2 -16783.633} C_VEL
LIN {X 0,Y 291.327,Z 362.823,A -85,B 0,C 180,E1 -16787.507,E2 -16787.507} C_VEL
LIN {X 0,Y 291.369,Z 362.798,A -85,B 0,C 180,E1 -16791.159,E2 -16791.159} C_VEL
LIN {X 0,Y 291.424,Z 362.979,A -85,B 0,C 180,E1 -16792.445,E2 -16792.445} C_VEL
LIN {X 0,Y 293.797,Z 372.059,A -85,B 0,C 180,E1 -16795.727,E2 -16795.727} C_VEL
LIN {X 0,Y 295.596,Z 375.854,A -85,B 0,C 180,E1 -16796.153,E2 -16796.153} C_VEL
LIN {X 0,Y 304.763,Z 394.811,A -85,B 0,C 180,E1 -16797.821,E2 -16797.821} C_VEL
LIN {X 0,Y 310.781,Z 409.403,A -85,B 0,C 180,E1 -16798.903,E2 -16798.903} C_VEL
LIN {X 0,Y 312.125,Z 417.826,A -85,B 0,C 180,E1 -16799.273,E2 -16799.273} C_VEL
LIN {X 0,Y 309.582,Z 496.705,A -85,B 0,C 180,E1 -16801.063,E2 -16801.063} C_VEL
LIN {X 0,Y 308.883,Z 512.958,A -85,B 0,C 180,E1 -16801.502,E2 -16801.502} C_VEL
LIN {X 0,Y 307.673,Z 527.195,A -85,B 0,C 180,E1 -16802.123,E2 -16802.123} C_VEL
LIN {X 0,Y 306.2,Z 540.354,A -85,B 0,C 180,E1 -16802.95,E2 -16802.95} C_VEL
LIN {X 0,Y 304.33,Z 554.09,A -85,B 0,C 180,E1 -16804.106,E2 -16804.106} C_VEL
LIN {X 0,Y 302.344,Z 566.419,A -85,B 0,C 180,E1 -16805.447,E2 -16805.447} C_VEL
LIN {X 0,Y 300.076,Z 578.462,A -85,B 0,C 180,E1 -16807.083,E2 -16807.083} C_VEL
LIN {X 0,Y 297.812,Z 589.317,A -85,B 0,C 180,E1 -16808.905,E2 -16808.905} C_VEL
LIN {X 0,Y 295.712,Z 599.092,A -85,B 0,C 180,E1 -16810.924,E2 -16810.924} C_VEL
LIN {X 0,Y 293.853,Z 607.578,A -85,B 0,C 180,E1 -16813.072,E2 -16813.072} C_VEL
LIN {X 0,Y 292.471,Z 614.966,A -85,B 0,C 180,E1 -16815.384,E2 -16815.384} C_VEL
LIN {X 0,Y 291.224,Z 620.393,A -85,B 0,C 180,E1 -16817.454,E2 -16817.454} C_VEL
LIN {X 0,Y 290.256,Z 626.097,A -85,B 0,C 180,E1 -16820.24,E2 -16820.24} C_VEL
LIN {X 0,Y 289.674,Z 630.241,A -85,B 0,C 180,E1 -16823.031,E2 -16823.031} C_VEL
LIN {X 0,Y 289.418,Z 632.955,A -85,B 0,C 180,E1 -16825.821,E2 -16825.821} C_VEL
LIN {X 0,Y 289.372,Z 634.316,A -85,B 0,C 180,E1 -16828.607,E2 -16828.607} C_VEL
LIN {X 0,Y 289.372,Z 634.349,A -85,B 0,C 180,E1 -16831.39,E2 -16831.39} C_VEL
LIN {X 0,Y 289.415,Z 633.052,A -85,B 0,C 180,E1 -16834.176,E2 -16834.176} C_VEL
LIN {X 0,Y 289.672,Z 630.395,A -85,B 0,C 180,E1 -16836.966,E2 -16836.966} C_VEL
LIN {X 0,Y 290.246,Z 626.305,A -85,B 0,C 180,E1 -16839.757,E2 -16839.757} C_VEL
LIN {X 0,Y 291.187,Z 620.661,A -85,B 0,C 180,E1 -16842.544,E2 -16842.544} C_VEL
LIN {X 0,Y 292.642,Z 614.294,A -85,B 0,C 180,E1 -16844.959,E2 -16844.959} C_VEL
LIN {X 0,Y 294.151,Z 606.624,A -85,B 0,C 180,E1 -16847.303,E2 -16847.303} C_VEL
LIN {X 0,Y 295.989,Z 598.098,A -85,B 0,C 180,E1 -16849.414,E2 -16849.414} C_VEL
LIN {X 0,Y 298.128,Z 588.125,A -85,B 0,C 180,E1 -16851.43,E2 -16851.43} C_VEL
LIN {X 0,Y 300.394,Z 577.022,A -85,B 0,C 180,E1 -16853.252,E2 -16853.252} C_VEL
LIN {X 0,Y 302.505,Z 565.974,A -85,B 0,C 180,E1 -16854.718,E2 -16854.718} C_VEL
LIN {X 0,Y 304.433,Z 553.976,A -85,B 0,C 180,E1 -16856.014,E2 -16856.014} C_VEL
LIN {X 0,Y 306.193,Z 540.696,A -85,B 0,C 180,E1 -16857.139,E2 -16857.139} C_VEL
LIN {X 0,Y 307.734,Z 526.893,A -85,B 0,C 180,E1 -16858.007,E2 -16858.007} C_VEL
LIN {X 0,Y 308.933,Z 512.518,A -85,B 0,C 180,E1 -16858.628,E2 -16858.628} C_VEL
LIN {X 0,Y 309.813,Z 492.443,A -85,B 0,C 180,E1 -16859.142,E2 -16859.142} C_VEL
LIN {X 0,Y 311.861,Z 427.564,A -85,B 0,C 180,E1 -16860.619,E2 -16860.619} C_VEL
LIN {X 0,Y 311.577,Z 423.715,A -85,B 0,C 180,E1 -16860.751,E2 -16860.751} C_VEL
LIN {X 0,Y 310.009,Z 418.264,A -85,B 0,C 180,E1 -16861.067,E2 -16861.067} C_VEL
LIN {X 0,Y 307.585,Z 413.25,A -85,B 0,C 180,E1 -16861.474,E2 -16861.474} C_VEL
LIN {X 0,Y 300.109,Z 400.059,A -85,B 0,C 180,E1 -16862.717,E2 -16862.717} C_VEL
LIN {X 0,Y 292.055,Z 383.017,A -85,B 0,C 180,E1 -16864.232,E2 -16864.232} C_VEL
LIN {X 0,Y 286.656,Z 372.389,A -85,B 0,C 180,E1 -16865.326,E2 -16865.326} C_VEL
LIN {X 0,Y 285.081,Z 366.506,A -85,B 0,C 180,E1 -16867.42,E2 -16867.42} C_VEL
LIN {X 0,Y 284.35,Z 363.735,A -85,B 0,C 180,E1 -16868.584,E2 -16868.584} C_VEL
LIN {X 0,Y 284.349,Z 363.691,A -85,B 0,C 180,E1 -16872.142,E2 -16872.142} C_VEL
LIN {X 0,Y 284.348,Z 363.661,A -85,B 0,C 180,E1 -16876.207,E2 -16876.207} C_VEL
LIN {X 0,Y 284.344,Z 363.67,A -85,B 0,C 180,E1 -16880.012,E2 -16880.012} C_VEL
LIN {X 0,Y 284.344,Z 363.654,A -85,B 0,C 180,E1 -16883.616,E2 -16883.616} C_VEL
LIN {X 0,Y 284.3,Z 363.693,A -85,B 0,C 180,E1 -16887.188,E2 -16887.188} C_VEL
LIN {X 0,Y 284.35,Z 363.63,A -85,B 0,C 180,E1 -16890.375,E2 -16890.375} C_VEL
LIN {X 0,Y 284.369,Z 363.66,A -85,B 0,C 180,E1 -16893.586,E2 -16893.586} C_VEL
LIN {X 0,Y 284.358,Z 363.689,A -85,B 0,C 180,E1 -16896.706,E2 -16896.706} C_VEL
LIN {X 0,Y 284.394,Z 363.684,A -85,B 0,C 180,E1 -16901.261,E2 -16901.261} C_VEL
LIN {X 0,Y 284.482,Z 363.651,A -85,B 0,C 180,E1 -16904.459,E2 -16904.459} C_VEL
LIN {X 0,Y 284.48,Z 363.666,A -85,B 0,C 180,E1 -16908.601,E2 -16908.601} C_VEL
LIN {X 0,Y 284.649,Z 363.634,A -85,B 0,C 180,E1 -16911.481,E2 -16911.481} C_VEL
LIN {X 0,Y 284.593,Z 363.657,A -85,B 0,C 180,E1 -16914.331,E2 -16914.331} C_VEL
LIN {X 0,Y 284.848,Z 363.62,A -85,B 0,C 180,E1 -16918.586,E2 -16918.586} C_VEL
LIN {X 0,Y 284.848,Z 363.62,A -85,B 0,C 180,E1 -16921.414,E2 -16921.414} C_VEL
LIN {X 0,Y 284.688,Z 363.644,A -85,B 0,C 180,E1 -16927.09,E2 -16927.09} C_VEL
LIN {X 0,Y 284.557,Z 363.64,A -85,B 0,C 180,E1 -16929.956,E2 -16929.956} C_VEL
LIN {X 0,Y 284.472,Z 363.659,A -85,B 0,C 180,E1 -16934.303,E2 -16934.303} C_VEL
LIN {X 0,Y 284.415,Z 363.671,A -85,B 0,C 180,E1 -16937.249,E2 -16937.249} C_VEL
LIN {X 0,Y 284.369,Z 363.673,A -85,B 0,C 180,E1 -16940.243,E2 -16940.243} C_VEL
LIN {X 0,Y 284.36,Z 363.688,A -85,B 0,C 180,E1 -16943.876,E2 -16943.876} C_VEL
LIN {X 0,Y 284.38,Z 363.641,A -85,B 0,C 180,E1 -16947.172,E2 -16947.172} C_VEL
LIN {X 0,Y 284.278,Z 363.663,A -85,B 0,C 180,E1 -16951.276,E2 -16951.276} C_VEL
LIN {X 0,Y 284.353,Z 363.672,A -85,B 0,C 180,E1 -16955.355,E2 -16955.355} C_VEL
LIN {X 0,Y 284.325,Z 363.646,A -85,B 0,C 180,E1 -16958.167,E2 -16958.167} C_VEL
LIN {X 0,Y 284.349,Z 363.688,A -85,B 0,C 180,E1 -16962.145,E2 -16962.145} C_VEL
LIN {X 0,Y 284.346,Z 363.667,A -85,B 0,C 180,E1 -16966.21,E2 -16966.21} C_VEL
LIN {X 0,Y 284.345,Z 363.667,A -85,B 0,C 180,E1 -16970.015,E2 -16970.015} C_VEL
LIN {X 0,Y 284.35,Z 363.794,A -85,B 0,C 180,E1 -16971.501,E2 -16971.501} C_VEL
LIN {X 0,Y 286.561,Z 372.015,A -85,B 0,C 180,E1 -16974.649,E2 -16974.649} C_VEL
LIN {X 0,Y 288.379,Z 375.866,A -85,B 0,C 180,E1 -16975.102,E2 -16975.102} C_VEL
LIN {X 0,Y 296.382,Z 391.801,A -85,B 0,C 180,E1 -16976.629,E2 -16976.629} C_VEL
LIN {X 0,Y 303.488,Z 408.147,A -85,B 0,C 180,E1 -16977.958,E2 -16977.958} C_VEL
LIN {X 0,Y 305.068,Z 412.53,A -85,B 0,C 180,E1 -16978.262,E2 -16978.262} C_VEL
LIN {X 0,Y 306.086,Z 418.657,A -85,B 0,C 180,E1 -16978.545,E2 -16978.545} C_VEL
LIN {X 0,Y 302.973,Z 509.118,A -85,B 0,C 180,E1 -16980.66,E2 -16980.66} C_VEL
LIN {X 0,Y 301.801,Z 523.877,A -85,B 0,C 180,E1 -16981.25,E2 -16981.25} C_VEL
LIN {X 0,Y 300.229,Z 537.893,A -85,B 0,C 180,E1 -16982.086,E2 -16982.086} C_VEL
LIN {X 0,Y 298.628,Z 550.026,A -85,B 0,C 180,E1 -16983.064,E2 -16983.064} C_VEL
LIN {X 0,Y 296.67,Z 562.268,A -85,B 0,C 180,E1 -16984.316,E2 -16984.316} C_VEL
LIN {X 0,Y 294.464,Z 574.407,A -85,B 0,C 180,E1 -16985.877,E2 -16985.877} C_VEL
LIN {X 0,Y 291.95,Z 586.019,A -85,B 0,C 180,E1 -16987.721,E2 -16987.721} C_VEL
LIN {X 0,Y 289.683,Z 596.402,A -85,B 0,C 180,E1 -16989.776,E2 -16989.776} C_VEL
LIN {X 0,Y 287.632,Z 605.1,A -85,B 0,C 180,E1 -16991.887,E2 -16991.887} C_VEL
LIN {X 0,Y 285.946,Z 613.162,A -85,B 0,C 180,E1 -16994.316,E2 -16994.316} C_VEL
LIN {X 0,Y 284.66,Z 618.899,A -85,B 0,C 180,E1 -16996.437,E2 -16996.437} C_VEL
LIN {X 0,Y 283.685,Z 623.596,A -85,B 0,C 180,E1 -16998.571,E2 -16998.571} C_VEL
LIN {X 0,Y 282.871,Z 628.468,A -85,B 0,C 180,E1 -17001.429,E2 -17001.429} C_VEL
LIN {X 0,Y 282.475,Z 631.946,A -85,B 0,C 180,E1 -17004.385,E2 -17004.385} C_VEL
LIN {X 0,Y 282.307,Z 633.845,A -85,B 0,C 180,E1 -17007.148,E2 -17007.148} C_VEL
LIN {X 0,Y 282.274,Z 634.5,A -85,B 0,C 180,E1 -17010.002,E2 -17010.002} C_VEL
LIN {X 0,Y 282.306,Z 633.828,A -85,B 0,C 180,E1 -17012.856,E2 -17012.856} C_VEL
LIN {X 0,Y 282.327,Z 633.008,A -85,B 0,C 180,E1 -17014.285,E2 -17014.285} C_VEL
LIN {X 0,Y 282.444,Z 632.831,A -85,B 0,C 180,E1 -17015.714,E2 -17015.714} C_VEL
LIN {X 0,Y 282.724,Z 632.221,A -85,B 0,C 180,E1 -17017.142,E2 -17017.142} C_VEL
LIN {X 0,Y 283.008,Z 631.215,A -85,B 0,C 180,E1 -17018.571,E2 -17018.571} C_VEL
LIN {X 0,Y 283.481,Z 629.797,A -85,B 0,C 180,E1 -17019.996,E2 -17019.996} C_VEL
LIN {X 0,Y 284.343,Z 626.819,A -85,B 0,C 180,E1 -17022.129,E2 -17022.129} C_VEL
LIN {X 0,Y 285.637,Z 622.813,A -85,B 0,C 180,E1 -17024.245,E2 -17024.245} C_VEL
LIN {X 0,Y 287.195,Z 617.682,A -85,B 0,C 180,E1 -17026.347,E2 -17026.347} C_VEL
LIN {X 0,Y 289.115,Z 610.919,A -85,B 0,C 180,E1 -17028.551,E2 -17028.551} C_VEL
LIN {X 0,Y 291.238,Z 603.535,A -85,B 0,C 180,E1 -17030.483,E2 -17030.483} C_VEL
LIN {X 0,Y 293.734,Z 594.141,A -85,B 0,C 180,E1 -17032.51,E2 -17032.51} C_VEL
LIN {X 0,Y 296.698,Z 582.432,A -85,B 0,C 180,E1 -17034.491,E2 -17034.491} C_VEL
LIN {X 0,Y 299.227,Z 571.116,A -85,B 0,C 180,E1 -17036.034,E2 -17036.034} C_VEL
LIN {X 0,Y 301.55,Z 558.783,A -85,B 0,C 180,E1 -17037.409,E2 -17037.409} C_VEL
LIN {X 0,Y 303.838,Z 544.846,A -85,B 0,C 180,E1 -17038.59,E2 -17038.59} C_VEL
LIN {X 0,Y 305.646,Z 530.692,A -85,B 0,C 180,E1 -17039.488,E2 -17039.488} C_VEL
LIN {X 0,Y 309.531,Z 498.754,A -85,B 0,C 180,E1 -17040.96,E2 -17040.96} C_VEL
LIN {X 0,Y 318.238,Z 439.629,A -85,B 0,C 180,E1 -17043.465,E2 -17043.465} C_VEL
LIN {X 0,Y 320.418,Z 425.047,A -85,B 0,C 180,E1 -17044.082,E2 -17044.082} C_VEL
LIN {X 0,Y 319.239,Z 421.239,A -85,B 0,C 180,E1 -17044.918,E2 -17044.918} C_VEL
LIN {X 0,Y 317.184,Z 418.481,A -85,B 0,C 180,E1 -17046.109,E2 -17046.109} C_VEL
LIN {X 0,Y 316.024,Z 417.027,A -85,B 0,C 180,E1 -17046.904,E2 -17046.904} C_VEL
LIN {X 0,Y 314.501,Z 414.676,A -85,B 0,C 180,E1 -17048.735,E2 -17048.735} C_VEL
LIN {X 0,Y 313.472,Z 413.109,A -85,B 0,C 180,E1 -17050.557,E2 -17050.557} C_VEL
LIN {X 0,Y 312.67,Z 412.424,A -85,B 0,C 180,E1 -17052.403,E2 -17052.403} C_VEL
LIN {X 0,Y 312.068,Z 412.663,A -85,B 0,C 180,E1 -17054.28,E2 -17054.28} C_VEL
LIN {X 0,Y 311.779,Z 413.571,A -85,B 0,C 180,E1 -17056.166,E2 -17056.166} C_VEL
LIN {X 0,Y 311.753,Z 415.204,A -85,B 0,C 180,E1 -17058.069,E2 -17058.069} C_VEL
LIN {X 0,Y 311.904,Z 417.63,A -85,B 0,C 180,E1 -17060.007,E2 -17060.007} C_VEL
LIN {X 0,Y 312.176,Z 419.227,A -85,B 0,C 180,E1 -17060.923,E2 -17060.923} C_VEL
LIN {X 0,Y 314.593,Z 425.225,A -85,B 0,C 180,E1 -17063.252,E2 -17063.252} C_VEL
LIN {X 0,Y 316.832,Z 431.668,A -85,B 0,C 180,E1 -17064.974,E2 -17064.974} C_VEL
LIN {X 0,Y 318.055,Z 446.204,A -85,B 0,C 180,E1 -17066.831,E2 -17066.831} C_VEL
LIN {X 0,Y 318.896,Z 459.795,A -85,B 0,C 180,E1 -17068.237,E2 -17068.237} C_VEL
LIN {X 0,Y 319.004,Z 464.64,A -85,B 0,C 180,E1 -17068.643,E2 -17068.643} C_VEL
LIN {X 0,Y 309.981,Z 535.492,A -85,B 0,C 180,E1 -17071.614,E2 -17071.614} C_VEL
LIN {X 0,Y 307.598,Z 549.253,A -85,B 0,C 180,E1 -17072.44,E2 -17072.44} C_VEL
LIN {X 0,Y 304.969,Z 562.001,A -85,B 0,C 180,E1 -17073.481,E2 -17073.481} C_VEL
LIN {X 0,Y 301.897,Z 574.961,A -85,B 0,C 180,E1 -17074.859,E2 -17074.859} C_VEL
LIN {X 0,Y 298.752,Z 586.54,A -85,B 0,C 180,E1 -17076.427,E2 -17076.427} C_VEL
LIN {X 0,Y 295.86,Z 596.271,A -85,B 0,C 180,E1 -17078.074,E2 -17078.074} C_VEL
LIN {X 0,Y 292.837,Z 605.496,A -85,B 0,C 180,E1 -17080.002,E2 -17080.002} C_VEL
LIN {X 0,Y 290.278,Z 613.182,A -85,B 0,C 180,E1 -17082.02,E2 -17082.02} C_VEL
LIN {X 0,Y 288.383,Z 618.47,A -85,B 0,C 180,E1 -17083.724,E2 -17083.724} C_VEL
LIN {X 0,Y 286.658,Z 623.657,A -85,B 0,C 180,E1 -17085.808,E2 -17085.808} C_VEL
LIN {X 0,Y 285.093,Z 627.72,A -85,B 0,C 180,E1 -17087.905,E2 -17087.905} C_VEL
LIN {X 0,Y 283.903,Z 630.728,A -85,B 0,C 180,E1 -17090.021,E2 -17090.021} C_VEL
LIN {X 0,Y 283.34,Z 632.164,A -85,B 0,C 180,E1 -17091.441,E2 -17091.441} C_VEL
LIN {X 0,Y 282.649,Z 633.716,A -85,B 0,C 180,E1 -17094.049,E2 -17094.049} C_VEL
LIN {X 0,Y 282.422,Z 633.977,A -85,B 0,C 180,E1 -17095.719,E2 -17095.719} C_VEL
LIN {X 0,Y 282.338,Z 633.705,A -85,B 0,C 180,E1 -17097.146,E2 -17097.146} C_VEL
LIN {X 0,Y 282.306,Z 633.021,A -85,B 0,C 180,E1 -17098.574,E2 -17098.574} C_VEL
LIN {X 0,Y 282.28,Z 631.903,A -85,B 0,C 180,E1 -17100,E2 -17100} C_VEL
LIN {X 0,Y 282.335,Z 629.343,A -85,B 0,C 180,E1 -17102.14,E2 -17102.14} C_VEL
LIN {X 0,Y 282.458,Z 625.679,A -85,B 0,C 180,E1 -17104.281,E2 -17104.281} C_VEL
LIN {X 0,Y 282.577,Z 620.771,A -85,B 0,C 180,E1 -17106.426,E2 -17106.426} C_VEL
LIN {X 0,Y 282.939,Z 614.521,A -85,B 0,C 180,E1 -17108.571,E2 -17108.571} C_VEL
LIN {X 0,Y 283.412,Z 606.695,A -85,B 0,C 180,E1 -17110.719,E2 -17110.719} C_VEL
LIN {X 0,Y 284.152,Z 596.844,A -85,B 0,C 180,E1 -17112.862,E2 -17112.862} C_VEL
LIN {X 0,Y 285.012,Z 586.706,A -85,B 0,C 180,E1 -17114.64,E2 -17114.64} C_VEL
LIN {X 0,Y 286.033,Z 574.659,A -85,B 0,C 180,E1 -17116.337,E2 -17116.337} C_VEL
LIN {X 0,Y 286.904,Z 562.875,A -85,B 0,C 180,E1 -17117.646,E2 -17117.646} C_VEL
LIN {X 0,Y 287.771,Z 549.72,A -85,B 0,C 180,E1 -17118.788,E2 -17118.788} C_VEL
LIN {X 0,Y 288.597,Z 535.084,A -85,B 0,C 180,E1 -17119.702,E2 -17119.702} C_VEL
LIN {X 0,Y 289.188,Z 519.347,A -85,B 0,C 180,E1 -17120.355,E2 -17120.355} C_VEL
LIN {X 0,Y 291.52,Z 452.829,A -85,B 0,C 180,E1 -17122.805,E2 -17122.805} C_VEL
LIN {X 0,Y 288.698,Z 424.326,A -85,B 0,C 180,E1 -17124.006,E2 -17124.006} C_VEL
LIN {X 0,Y 288.497,Z 419.982,A -85,B 0,C 180,E1 -17124.228,E2 -17124.228} C_VEL
LIN {X 0,Y 290.127,Z 401.708,A -85,B 0,C 180,E1 -17127.795,E2 -17127.795} C_VEL
LIN {X 0,Y 290.934,Z 393.859,A -85,B 0,C 180,E1 -17129.326,E2 -17129.326} C_VEL
LIN {X 0,Y 287.845,Z 379.218,A -85,B 0,C 180,E1 -17132.49,E2 -17132.49} C_VEL
LIN {X 0,Y 284.392,Z 363.836,A -85,B 0,C 180,E1 -17135.973,E2 -17135.973} C_VEL
LIN {X 0,Y 284.312,Z 363.696,A -85,B 0,C 180,E1 -17139.994,E2 -17139.994} C_VEL
LIN {X 0,Y 284.251,Z 363.671,A -85,B 0,C 180,E1 -17144.189,E2 -17144.189} C_VEL
LIN {X 0,Y 284.278,Z 363.699,A -85,B 0,C 180,E1 -17148.124,E2 -17148.124} C_VEL
LIN {X 0,Y 284.34,Z 363.815,A -85,B 0,C 180,E1 -17151.608,E2 -17151.608} C_VEL
LIN {X 0,Y 286.341,Z 371.255,A -85,B 0,C 180,E1 -17154.485,E2 -17154.485} C_VEL
LIN {X 0,Y 286.79,Z 372.74,A -85,B 0,C 180,E1 -17154.851,E2 -17154.851} C_VEL
LIN {X 0,Y 294.909,Z 388.863,A -85,B 0,C 180,E1 -17156.437,E2 -17156.437} C_VEL
LIN {X 0,Y 300.987,Z 402.185,A -85,B 0,C 180,E1 -17157.571,E2 -17157.571} C_VEL
LIN {X 0,Y 304.918,Z 412.018,A -85,B 0,C 180,E1 -17158.307,E2 -17158.307} C_VEL
LIN {X 0,Y 306.046,Z 418.503,A -85,B 0,C 180,E1 -17158.612,E2 -17158.612} C_VEL
LIN {X 0,Y 303.3,Z 498.551,A -85,B 0,C 180,E1 -17160.453,E2 -17160.453} C_VEL
LIN {X 0,Y 302.604,Z 514.114,A -85,B 0,C 180,E1 -17160.902,E2 -17160.902} C_VEL
LIN {X 0,Y 301.352,Z 527.968,A -85,B 0,C 180,E1 -17161.533,E2 -17161.533} C_VEL
LIN {X 0,Y 299.761,Z 541.486,A -85,B 0,C 180,E1 -17162.415,E2 -17162.415} C_VEL
LIN {X 0,Y 297.926,Z 554.214,A -85,B 0,C 180,E1 -17163.52,E2 -17163.52} C_VEL
LIN {X 0,Y 295.893,Z 566.423,A -85,B 0,C 180,E1 -17164.875,E2 -17164.875} C_VEL
LIN {X 0,Y 293.516,Z 578.466,A -85,B 0,C 180,E1 -17166.541,E2 -17166.541} C_VEL
LIN {X 0,Y 291.185,Z 589.32,A -85,B 0,C 180,E1 -17168.402,E2 -17168.402} C_VEL
LIN {X 0,Y 288.992,Z 599.094,A -85,B 0,C 180,E1 -17170.463,E2 -17170.463} C_VEL
LIN {X 0,Y 286.894,Z 608.155,A -85,B 0,C 180,E1 -17172.82,E2 -17172.82} C_VEL
LIN {X 0,Y 285.583,Z 614.968,A -85,B 0,C 180,E1 -17175.023,E2 -17175.023} C_VEL
LIN {X 0,Y 284.259,Z 620.395,A -85,B 0,C 180,E1 -17177.141,E2 -17177.141} C_VEL
LIN {X 0,Y 283.22,Z 626.098,A -85,B 0,C 180,E1 -17179.995,E2 -17179.995} C_VEL
LIN {X 0,Y 282.602,Z 630.241,A -85,B 0,C 180,E1 -17182.855,E2 -17182.855} C_VEL
LIN {X 0,Y 282.329,Z 632.956,A -85,B 0,C 180,E1 -17185.715,E2 -17185.715} C_VEL
LIN {X 0,Y 282.297,Z 634.316,A -85,B 0,C 180,E1 -17188.572,E2 -17188.572} C_VEL
LIN {X 0,Y 282.296,Z 634.348,A -85,B 0,C 180,E1 -17191.425,E2 -17191.425} C_VEL
LIN {X 0,Y 282.326,Z 633.051,A -85,B 0,C 180,E1 -17194.281,E2 -17194.281} C_VEL
LIN {X 0,Y 282.6,Z 630.394,A -85,B 0,C 180,E1 -17197.141,E2 -17197.141} C_VEL
LIN {X 0,Y 283.208,Z 626.304,A -85,B 0,C 180,E1 -17200.002,E2 -17200.002} C_VEL
LIN {X 0,Y 284.227,Z 620.659,A -85,B 0,C 180,E1 -17202.856,E2 -17202.856} C_VEL
LIN {X 0,Y 285.735,Z 614.293,A -85,B 0,C 180,E1 -17205.33,E2 -17205.33} C_VEL
LIN {X 0,Y 287.338,Z 606.622,A -85,B 0,C 180,E1 -17207.727,E2 -17207.727} C_VEL
LIN {X 0,Y 289.258,Z 598.096,A -85,B 0,C 180,E1 -17209.884,E2 -17209.884} C_VEL
LIN {X 0,Y 291.506,Z 588.122,A -85,B 0,C 180,E1 -17211.942,E2 -17211.942} C_VEL
LIN {X 0,Y 293.876,Z 577.019,A -85,B 0,C 180,E1 -17213.799,E2 -17213.799} C_VEL
LIN {X 0,Y 296.234,Z 564.796,A -85,B 0,C 180,E1 -17215.435,E2 -17215.435} C_VEL
LIN {X 0,Y 298.304,Z 552.213,A -85,B 0,C 180,E1 -17216.779,E2 -17216.779} C_VEL
LIN {X 0,Y 300.128,Z 538.429,A -85,B 0,C 180,E1 -17217.924,E2 -17217.924} C_VEL
LIN {X 0,Y 301.744,Z 524.598,A -85,B 0,C 180,E1 -17218.756,E2 -17218.756} C_VEL
LIN {X 0,Y 302.821,Z 511.364,A -85,B 0,C 180,E1 -17219.309,E2 -17219.309} C_VEL
LIN {X 0,Y 303.811,Z 487.052,A -85,B 0,C 180,E1 -17219.918,E2 -17219.918} C_VEL
LIN {X 0,Y 305.962,Z 417.451,A -85,B 0,C 180,E1 -17221.546,E2 -17221.546} C_VEL
LIN {X 0,Y 304.562,Z 410.91,A -85,B 0,C 180,E1 -17221.886,E2 -17221.886} C_VEL
LIN {X 0,Y 300.109,Z 400.059,A -85,B 0,C 180,E1 -17222.717,E2 -17222.717} C_VEL
LIN {X 0,Y 298.175,Z 397.06,A -85,B 0,C 180,E1 -17223.041,E2 -17223.041} C_VEL
LIN {X 0,Y 293.852,Z 393.288,A -85,B 0,C 180,E1 -17223.698,E2 -17223.698} C_VEL
LIN {X 0,Y 288.48,Z 388.93,A -85,B 0,C 180,E1 -17224.541,E2 -17224.541} C_VEL
LIN {X 0,Y 287.011,Z 387.077,A -85,B 0,C 180,E1 -17224.798,E2 -17224.798} C_VEL
LIN {X 0,Y 279.4,Z 372.297,A -85,B 0,C 180,E1 -17226.397,E2 -17226.397} C_VEL
LIN {X 0,Y 277.332,Z 364.781,A -85,B 0,C 180,E1 -17229.309,E2 -17229.309} C_VEL
LIN {X 0,Y 277.292,Z 364.554,A -85,B 0,C 180,E1 -17231.219,E2 -17231.219} C_VEL
LIN {X 0,Y 277.282,Z 364.535,A -85,B 0,C 180,E1 -17235.206,E2 -17235.206} C_VEL
LIN {X 0,Y 277.29,Z 364.56,A -85,B 0,C 180,E1 -17239.492,E2 -17239.492} C_VEL
LIN {X 0,Y 277.279,Z 364.523,A -85,B 0,C 180,E1 -17242.532,E2 -17242.532} C_VEL
LIN {X 0,Y 277.246,Z 364.578,A -85,B 0,C 180,E1 -17246.104,E2 -17246.104} C_VEL
LIN {X 0,Y 277.253,Z 364.522,A -85,B 0,C 180,E1 -17249.537,E2 -17249.537} C_VEL
LIN {X 0,Y 277.35,Z 364.516,A -85,B 0,C 180,E1 -17252.863,E2 -17252.863} C_VEL
LIN {X 0,Y 277.329,Z 364.565,A -85,B 0,C 180,E1 -17256.079,E2 -17256.079} C_VEL
LIN {X 0,Y 277.336,Z 364.559,A -85,B 0,C 180,E1 -17260.765,E2 -17260.765} C_VEL
LIN {X 0,Y 277.425,Z 364.533,A -85,B 0,C 180,E1 -17265.325,E2 -17265.325} C_VEL
LIN {X 0,Y 277.497,Z 364.522,A -85,B 0,C 180,E1 -17269.788,E2 -17269.788} C_VEL
LIN {X 0,Y 277.643,Z 364.519,A -85,B 0,C 180,E1 -17272.729,E2 -17272.729} C_VEL
LIN {X 0,Y 277.814,Z 364.496,A -85,B 0,C 180,E1 -17278.55,E2 -17278.55} C_VEL
LIN {X 0,Y 277.814,Z 364.496,A -85,B 0,C 180,E1 -17281.449,E2 -17281.449} C_VEL
LIN {X 0,Y 277.643,Z 364.52,A -85,B 0,C 180,E1 -17287.271,E2 -17287.271} C_VEL
LIN {X 0,Y 277.497,Z 364.52,A -85,B 0,C 180,E1 -17290.212,E2 -17290.212} C_VEL
LIN {X 0,Y 277.425,Z 364.532,A -85,B 0,C 180,E1 -17294.675,E2 -17294.675} C_VEL
LIN {X 0,Y 277.335,Z 364.558,A -85,B 0,C 180,E1 -17299.234,E2 -17299.234} C_VEL
LIN {X 0,Y 277.309,Z 364.567,A -85,B 0,C 180,E1 -17304.171,E2 -17304.171} C_VEL
LIN {X 0,Y 277.308,Z 364.514,A -85,B 0,C 180,E1 -17307.503,E2 -17307.503} C_VEL
LIN {X 0,Y 277.238,Z 364.522,A -85,B 0,C 180,E1 -17310.474,E2 -17310.474} C_VEL
LIN {X 0,Y 277.245,Z 364.577,A -85,B 0,C 180,E1 -17313.896,E2 -17313.896} C_VEL
LIN {X 0,Y 277.278,Z 364.523,A -85,B 0,C 180,E1 -17317.468,E2 -17317.468} C_VEL
LIN {X 0,Y 277.292,Z 364.57,A -85,B 0,C 180,E1 -17321.222,E2 -17321.222} C_VEL
LIN {X 0,Y 277.281,Z 364.536,A -85,B 0,C 180,E1 -17325.21,E2 -17325.21} C_VEL
LIN {X 0,Y 277.29,Z 364.547,A -85,B 0,C 180,E1 -17329.496,E2 -17329.496} C_VEL
LIN {X 0,Y 277.328,Z 364.706,A -85,B 0,C 180,E1 -17330.691,E2 -17330.691} C_VEL
LIN {X 0,Y 279.344,Z 372.159,A -85,B 0,C 180,E1 -17333.619,E2 -17333.619} C_VEL
LIN {X 0,Y 283.382,Z 379.985,A -85,B 0,C 180,E1 -17334.52,E2 -17334.52} C_VEL
LIN {X 0,Y 291.503,Z 396.384,A -85,B 0,C 180,E1 -17336.128,E2 -17336.128} C_VEL
LIN {X 0,Y 298.538,Z 412.809,A -85,B 0,C 180,E1 -17337.491,E2 -17337.491} C_VEL
LIN {X 0,Y 299.485,Z 416.199,A -85,B 0,C 180,E1 -17337.701,E2 -17337.701} C_VEL
LIN {X 0,Y 299.99,Z 420.281,A -85,B 0,C 180,E1 -17337.875,E2 -17337.875} C_VEL
LIN {X 0,Y 296.821,Z 509.133,A -85,B 0,C 180,E1 -17339.99,E2 -17339.99} C_VEL
LIN {X 0,Y 295.615,Z 523.886,A -85,B 0,C 180,E1 -17340.59,E2 -17340.59} C_VEL
LIN {X 0,Y 293.991,Z 537.9,A -85,B 0,C 180,E1 -17341.44,E2 -17341.44} C_VEL
LIN {X 0,Y 292.327,Z 550.031,A -85,B 0,C 180,E1 -17342.434,E2 -17342.434} C_VEL
LIN {X 0,Y 290.108,Z 563.243,A -85,B 0,C 180,E1 -17343.823,E2 -17343.823} C_VEL
LIN {X 0,Y 287.751,Z 575.583,A -85,B 0,C 180,E1 -17345.47,E2 -17345.47} C_VEL
LIN {X 0,Y 285.368,Z 586.022,A -85,B 0,C 180,E1 -17347.179,E2 -17347.179} C_VEL
LIN {X 0,Y 283.014,Z 596.404,A -85,B 0,C 180,E1 -17349.278,E2 -17349.278} C_VEL
LIN {X 0,Y 280.902,Z 604.968,A -85,B 0,C 180,E1 -17351.4,E2 -17351.4} C_VEL
LIN {X 0,Y 279.052,Z 613.163,A -85,B 0,C 180,E1 -17353.919,E2 -17353.919} C_VEL
LIN {X 0,Y 277.744,Z 618.9,A -85,B 0,C 180,E1 -17356.093,E2 -17356.093} C_VEL
LIN {X 0,Y 276.697,Z 623.598,A -85,B 0,C 180,E1 -17358.278,E2 -17358.278} C_VEL
LIN {X 0,Y 275.825,Z 628.469,A -85,B 0,C 180,E1 -17361.208,E2 -17361.208} C_VEL
LIN {X 0,Y 275.392,Z 631.851,A -85,B 0,C 180,E1 -17364.143,E2 -17364.143} C_VEL
LIN {X 0,Y 275.22,Z 633.845,A -85,B 0,C 180,E1 -17367.074,E2 -17367.074} C_VEL
LIN {X 0,Y 275.2,Z 634.5,A -85,B 0,C 180,E1 -17370.002,E2 -17370.002} C_VEL
LIN {X 0,Y 275.219,Z 633.827,A -85,B 0,C 180,E1 -17372.929,E2 -17372.929} C_VEL
LIN {X 0,Y 275.241,Z 633.007,A -85,B 0,C 180,E1 -17374.395,E2 -17374.395} C_VEL
LIN {X 0,Y 275.677,Z 632.477,A -85,B 0,C 180,E1 -17377.325,E2 -17377.325} C_VEL
LIN {X 0,Y 275.976,Z 631.572,A -85,B 0,C 180,E1 -17378.791,E2 -17378.791} C_VEL
LIN {X 0,Y 277.092,Z 628.549,A -85,B 0,C 180,E1 -17381.709,E2 -17381.709} C_VEL
LIN {X 0,Y 278.305,Z 625.117,A -85,B 0,C 180,E1 -17383.883,E2 -17383.883} C_VEL
LIN {X 0,Y 279.903,Z 620.633,A -85,B 0,C 180,E1 -17386.035,E2 -17386.035} C_VEL
LIN {X 0,Y 281.832,Z 614.706,A -85,B 0,C 180,E1 -17388.275,E2 -17388.275} C_VEL
LIN {X 0,Y 284.402,Z 606.803,A -85,B 0,C 180,E1 -17390.62,E2 -17390.62} C_VEL
LIN {X 0,Y 287.028,Z 598.136,A -85,B 0,C 180,E1 -17392.686,E2 -17392.686} C_VEL
LIN {X 0,Y 290.114,Z 587.506,A -85,B 0,C 180,E1 -17394.703,E2 -17394.703} C_VEL
LIN {X 0,Y 293.215,Z 575.552,A -85,B 0,C 180,E1 -17396.516,E2 -17396.516} C_VEL
LIN {X 0,Y 295.786,Z 564.04,A -85,B 0,C 180,E1 -17397.931,E2 -17397.931} C_VEL
LIN {X 0,Y 298.246,Z 551.828,A -85,B 0,C 180,E1 -17399.11,E2 -17399.11} C_VEL
LIN {X 0,Y 300.338,Z 538.898,A -85,B 0,C 180,E1 -17400.1,E2 -17400.1} C_VEL
LIN {X 0,Y 302.538,Z 521.933,A -85,B 0,C 180,E1 -17401.027,E2 -17401.027} C_VEL
LIN {X 0,Y 306.488,Z 494.106,A -85,B 0,C 180,E1 -17402.268,E2 -17402.268} C_VEL
LIN {X 0,Y 316.855,Z 428.397,A -85,B 0,C 180,E1 -17405.114,E2 -17405.114} C_VEL
LIN {X 0,Y 316.171,Z 426.752,A -85,B 0,C 180,E1 -17405.587,E2 -17405.587} C_VEL
LIN {X 0,Y 313.107,Z 422.842,A -85,B 0,C 180,E1 -17407.624,E2 -17407.624} C_VEL
LIN {X 0,Y 310.42,Z 419.791,A -85,B 0,C 180,E1 -17410.062,E2 -17410.062} C_VEL
LIN {X 0,Y 309.353,Z 418.776,A -85,B 0,C 180,E1 -17411.435,E2 -17411.435} C_VEL
LIN {X 0,Y 308.46,Z 418.396,A -85,B 0,C 180,E1 -17413.19,E2 -17413.19} C_VEL
LIN {X 0,Y 307.978,Z 418.929,A -85,B 0,C 180,E1 -17415.027,E2 -17415.027} C_VEL
LIN {X 0,Y 308.304,Z 421.137,A -85,B 0,C 180,E1 -17417.704,E2 -17417.704} C_VEL
LIN {X 0,Y 309.551,Z 424.603,A -85,B 0,C 180,E1 -17420.026,E2 -17420.026} C_VEL
LIN {X 0,Y 311.602,Z 430.068,A -85,B 0,C 180,E1 -17422.341,E2 -17422.341} C_VEL
LIN {X 0,Y 313.602,Z 436.157,A -85,B 0,C 180,E1 -17424.135,E2 -17424.135} C_VEL
LIN {X 0,Y 314.395,Z 448.742,A -85,B 0,C 180,E1 -17425.804,E2 -17425.804} C_VEL
LIN {X 0,Y 314.973,Z 462.105,A -85,B 0,C 180,E1 -17427.254,E2 -17427.254} C_VEL
LIN {X 0,Y 314.911,Z 466.826,A -85,B 0,C 180,E1 -17427.643,E2 -17427.643} C_VEL
LIN {X 0,Y 305.463,Z 535.605,A -85,B 0,C 180,E1 -17430.589,E2 -17430.589} C_VEL
LIN {X 0,Y 302.951,Z 549.173,A -85,B 0,C 180,E1 -17431.415,E2 -17431.415} C_VEL
LIN {X 0,Y 299.776,Z 563.415,A -85,B 0,C 180,E1 -17432.607,E2 -17432.607} C_VEL
LIN {X 0,Y 296.521,Z 575.952,A -85,B 0,C 180,E1 -17433.993,E2 -17433.993} C_VEL
LIN {X 0,Y 293.185,Z 587.286,A -85,B 0,C 180,E1 -17435.575,E2 -17435.575} C_VEL
LIN {X 0,Y 289.712,Z 597.958,A -85,B 0,C 180,E1 -17437.462,E2 -17437.462} C_VEL
LIN {X 0,Y 286.869,Z 605.915,A -85,B 0,C 180,E1 -17439.192,E2 -17439.192} C_VEL
LIN {X 0,Y 284.016,Z 613.482,A -85,B 0,C 180,E1 -17441.235,E2 -17441.235} C_VEL
LIN {X 0,Y 282.281,Z 617.733,A -85,B 0,C 180,E1 -17442.617,E2 -17442.617} C_VEL
LIN {X 0,Y 280.346,Z 623.033,A -85,B 0,C 180,E1 -17444.739,E2 -17444.739} C_VEL
LIN {X 0,Y 278.694,Z 627.204,A -85,B 0,C 180,E1 -17446.882,E2 -17446.882} C_VEL
LIN {X 0,Y 277.748,Z 629.421,A -85,B 0,C 180,E1 -17448.321,E2 -17448.321} C_VEL
LIN {X 0,Y 276.919,Z 631.157,A -85,B 0,C 180,E1 -17449.767,E2 -17449.767} C_VEL
LIN {X 0,Y 276.312,Z 632.485,A -85,B 0,C 180,E1 -17451.222,E2 -17451.222} C_VEL
LIN {X 0,Y 275.872,Z 633.404,A -85,B 0,C 180,E1 -17452.682,E2 -17452.682} C_VEL
LIN {X 0,Y 275.536,Z 633.871,A -85,B 0,C 180,E1 -17454.144,E2 -17454.144} C_VEL
LIN {X 0,Y 275.339,Z 633.915,A -85,B 0,C 180,E1 -17455.608,E2 -17455.608} C_VEL
LIN {X 0,Y 275.253,Z 633.552,A -85,B 0,C 180,E1 -17457.073,E2 -17457.073} C_VEL
LIN {X 0,Y 275.233,Z 632.759,A -85,B 0,C 180,E1 -17458.537,E2 -17458.537} C_VEL
LIN {X 0,Y 275.205,Z 631.488,A -85,B 0,C 180,E1 -17460,E2 -17460} C_VEL
LIN {X 0,Y 275.269,Z 628.752,A -85,B 0,C 180,E1 -17462.195,E2 -17462.195} C_VEL
LIN {X 0,Y 275.383,Z 624.889,A -85,B 0,C 180,E1 -17464.391,E2 -17464.391} C_VEL
LIN {X 0,Y 275.53,Z 619.787,A -85,B 0,C 180,E1 -17466.591,E2 -17466.591} C_VEL
LIN {X 0,Y 275.9,Z 613.323,A -85,B 0,C 180,E1 -17468.792,E2 -17468.792} C_VEL
LIN {X 0,Y 276.423,Z 605.143,A -85,B 0,C 180,E1 -17470.993,E2 -17470.993} C_VEL
LIN {X 0,Y 277.044,Z 596.798,A -85,B 0,C 180,E1 -17472.825,E2 -17472.825} C_VEL
LIN {X 0,Y 277.899,Z 586.666,A -85,B 0,C 180,E1 -17474.649,E2 -17474.649} C_VEL
LIN {X 0,Y 278.887,Z 575.289,A -85,B 0,C 180,E1 -17476.303,E2 -17476.303} C_VEL
LIN {X 0,Y 279.824,Z 562.912,A -85,B 0,C 180,E1 -17477.73,E2 -17477.73} C_VEL
LIN {X 0,Y 280.699,Z 549.838,A -85,B 0,C 180,E1 -17478.9,E2 -17478.9} C_VEL
LIN {X 0,Y 281.528,Z 535.312,A -85,B 0,C 180,E1 -17479.838,E2 -17479.838} C_VEL
LIN {X 0,Y 282.135,Z 519.755,A -85,B 0,C 180,E1 -17480.506,E2 -17480.506} C_VEL
LIN {X 0,Y 284.526,Z 453.226,A -85,B 0,C 180,E1 -17483.056,E2 -17483.056} C_VEL
LIN {X 0,Y 281.74,Z 424.681,A -85,B 0,C 180,E1 -17484.304,E2 -17484.304} C_VEL
LIN {X 0,Y 281.534,Z 420.073,A -85,B 0,C 180,E1 -17484.52,E2 -17484.52} C_VEL
LIN {X 0,Y 283.207,Z 401.858,A -85,B 0,C 180,E1 -17488.132,E2 -17488.132} C_VEL
LIN {X 0,Y 283.88,Z 394.085,A -85,B 0,C 180,E1 -17489.679,E2 -17489.679} C_VEL
LIN {X 0,Y 280.308,Z 377.877,A -85,B 0,C 180,E1 -17493.274,E2 -17493.274} C_VEL
LIN {X 0,Y 277.376,Z 364.696,A -85,B 0,C 180,E1 -17496.335,E2 -17496.335} C_VEL
LIN {X 0,Y 277.228,Z 364.576,A -85,B 0,C 180,E1 -17500.487,E2 -17500.487} C_VEL
LIN {X 0,Y 277.206,Z 364.546,A -85,B 0,C 180,E1 -17504.773,E2 -17504.773} C_VEL
LIN {X 0,Y 277.216,Z 364.567,A -85,B 0,C 180,E1 -17508.763,E2 -17508.763} C_VEL
LIN {X 0,Y 277.313,Z 364.609,A -85,B 0,C 180,E1 -17510.683,E2 -17510.683} C_VEL
LIN {X 0,Y 277.862,Z 366.697,A -85,B 0,C 180,E1 -17511.637,E2 -17511.637} C_VEL
LIN {X 0,Y 279.362,Z 372.253,A -85,B 0,C 180,E1 -17513.723,E2 -17513.723} C_VEL
LIN {X 0,Y 286.088,Z 385.23,A -85,B 0,C 180,E1 -17515.146,E2 -17515.146} C_VEL
LIN {X 0,Y 294.191,Z 402.454,A -85,B 0,C 180,E1 -17516.733,E2 -17516.733} C_VEL
LIN {X 0,Y 299.162,Z 414.75,A -85,B 0,C 180,E1 -17517.699,E2 -17517.699} C_VEL
LIN {X 0,Y 299.941,Z 420.494,A -85,B 0,C 180,E1 -17517.952,E2 -17517.952} C_VEL
LIN {X 0,Y 296.714,Z 509.649,A -85,B 0,C 180,E1 -17520.075,E2 -17520.075} C_VEL
LIN {X 0,Y 295.494,Z 524.168,A -85,B 0,C 180,E1 -17520.671,E2 -17520.671} C_VEL
LIN {X 0,Y 293.894,Z 538.111,A -85,B 0,C 180,E1 -17521.524,E2 -17521.524} C_VEL
LIN {X 0,Y 292.081,Z 551.071,A -85,B 0,C 180,E1 -17522.599,E2 -17522.599} C_VEL
LIN {X 0,Y 289.922,Z 563.88,A -85,B 0,C 180,E1 -17523.967,E2 -17523.967} C_VEL
LIN {X 0,Y 287.518,Z 576.275,A -85,B 0,C 180,E1 -17525.637,E2 -17525.637} C_VEL
LIN {X 0,Y 285.018,Z 587.542,A -85,B 0,C 180,E1 -17527.528,E2 -17527.528} C_VEL
LIN {X 0,Y 282.644,Z 597.612,A -85,B 0,C 180,E1 -17529.626,E2 -17529.626} C_VEL
LIN {X 0,Y 280.612,Z 605.974,A -85,B 0,C 180,E1 -17531.754,E2 -17531.754} C_VEL
LIN {X 0,Y 278.897,Z 613.962,A -85,B 0,C 180,E1 -17534.281,E2 -17534.281} C_VEL
LIN {X 0,Y 277.313,Z 620.396,A -85,B 0,C 180,E1 -17536.814,E2 -17536.814} C_VEL
LIN {X 0,Y 276.205,Z 626.099,A -85,B 0,C 180,E1 -17539.738,E2 -17539.738} C_VEL
LIN {X 0,Y 275.53,Z 630.242,A -85,B 0,C 180,E1 -17542.671,E2 -17542.671} C_VEL
LIN {X 0,Y 275.243,Z 632.956,A -85,B 0,C 180,E1 -17545.605,E2 -17545.605} C_VEL
LIN {X 0,Y 275.223,Z 634.317,A -85,B 0,C 180,E1 -17548.535,E2 -17548.535} C_VEL
LIN {X 0,Y 275.223,Z 634.348,A -85,B 0,C 180,E1 -17551.461,E2 -17551.461} C_VEL
LIN {X 0,Y 275.242,Z 633.051,A -85,B 0,C 180,E1 -17554.391,E2 -17554.391} C_VEL
LIN {X 0,Y 275.528,Z 630.393,A -85,B 0,C 180,E1 -17557.325,E2 -17557.325} C_VEL
LIN {X 0,Y 276.193,Z 626.303,A -85,B 0,C 180,E1 -17560.258,E2 -17560.258} C_VEL
LIN {X 0,Y 277.284,Z 620.658,A -85,B 0,C 180,E1 -17563.184,E2 -17563.184} C_VEL
LIN {X 0,Y 278.818,Z 614.291,A -85,B 0,C 180,E1 -17565.72,E2 -17565.72} C_VEL
LIN {X 0,Y 280.598,Z 606.374,A -85,B 0,C 180,E1 -17568.243,E2 -17568.243} C_VEL
LIN {X 0,Y 282.562,Z 598.093,A -85,B 0,C 180,E1 -17570.376,E2 -17570.376} C_VEL
LIN {X 0,Y 284.887,Z 588.119,A -85,B 0,C 180,E1 -17572.479,E2 -17572.479} C_VEL
LIN {X 0,Y 287.393,Z 577.015,A -85,B 0,C 180,E1 -17574.37,E2 -17574.37} C_VEL
LIN {X 0,Y 289.859,Z 564.568,A -85,B 0,C 180,E1 -17576.066,E2 -17576.066} C_VEL
LIN {X 0,Y 291.966,Z 552.207,A -85,B 0,C 180,E1 -17577.408,E2 -17577.408} C_VEL
LIN {X 0,Y 293.892,Z 538.421,A -85,B 0,C 180,E1 -17578.57,E2 -17578.57} C_VEL
LIN {X 0,Y 295.543,Z 524.588,A -85,B 0,C 180,E1 -17579.418,E2 -17579.418} C_VEL
LIN {X 0,Y 296.664,Z 511.348,A -85,B 0,C 180,E1 -17579.979,E2 -17579.979} C_VEL
LIN {X 0,Y 297.749,Z 485.238,A -85,B 0,C 180,E1 -17580.641,E2 -17580.641} C_VEL
LIN {X 0,Y 299.908,Z 418.627,A -85,B 0,C 180,E1 -17582.226,E2 -17582.226} C_VEL
LIN {X 0,Y 298.697,Z 413.246,A -85,B 0,C 180,E1 -17582.522,E2 -17582.522} C_VEL
LIN {X 0,Y 292.015,Z 397.569,A -85,B 0,C 180,E1 -17583.815,E2 -17583.815} C_VEL
LIN {X 0,Y 287.011,Z 387.077,A -85,B 0,C 180,E1 -17584.798,E2 -17584.798} C_VEL
LIN {X 0,Y 284.7,Z 384.481,A -85,B 0,C 180,E1 -17585.201,E2 -17585.201} C_VEL
LIN {X 0,Y 275.636,Z 377.99,A -85,B 0,C 180,E1 -17586.746,E2 -17586.746} C_VEL
LIN {X 0,Y 273.586,Z 375.224,A -85,B 0,C 180,E1 -17587.156,E2 -17587.156} C_VEL
LIN {X 0,Y 272.068,Z 372.071,A -85,B 0,C 180,E1 -17587.582,E2 -17587.582} C_VEL
LIN {X 0,Y 270.279,Z 365.545,A -85,B 0,C 180,E1 -17590.304,E2 -17590.304} C_VEL
LIN {X 0,Y 270.225,Z 365.416,A -85,B 0,C 180,E1 -17594.602,E2 -17594.602} C_VEL
LIN {X 0,Y 270.264,Z 365.443,A -85,B 0,C 180,E1 -17598.945,E2 -17598.945} C_VEL
LIN {X 0,Y 270.233,Z 365.405,A -85,B 0,C 180,E1 -17603.261,E2 -17603.261} C_VEL
LIN {X 0,Y 270.196,Z 365.454,A -85,B 0,C 180,E1 -17606.891,E2 -17606.891} C_VEL
LIN {X 0,Y 270.188,Z 365.391,A -85,B 0,C 180,E1 -17610.382,E2 -17610.382} C_VEL
LIN {X 0,Y 270.257,Z 365.418,A -85,B 0,C 180,E1 -17613.763,E2 -17613.763} C_VEL
LIN {X 0,Y 270.228,Z 365.443,A -85,B 0,C 180,E1 -17617.038,E2 -17617.038} C_VEL
LIN {X 0,Y 270.292,Z 365.432,A -85,B 0,C 180,E1 -17620.244,E2 -17620.244} C_VEL
LIN {X 0,Y 270.393,Z 365.406,A -85,B 0,C 180,E1 -17624.935,E2 -17624.935} C_VEL
LIN {X 0,Y 270.432,Z 365.404,A -85,B 0,C 180,E1 -17629.518,E2 -17629.518} C_VEL
LIN {X 0,Y 270.601,Z 365.396,A -85,B 0,C 180,E1 -17632.538,E2 -17632.538} C_VEL
LIN {X 0,Y 270.779,Z 365.372,A -85,B 0,C 180,E1 -17638.513,E2 -17638.513} C_VEL
LIN {X 0,Y 270.78,Z 365.372,A -85,B 0,C 180,E1 -17641.487,E2 -17641.487} C_VEL
LIN {X 0,Y 270.601,Z 365.396,A -85,B 0,C 180,E1 -17647.461,E2 -17647.461} C_VEL
LIN {X 0,Y 270.432,Z 365.402,A -85,B 0,C 180,E1 -17650.481,E2 -17650.481} C_VEL
LIN {X 0,Y 270.393,Z 365.404,A -85,B 0,C 180,E1 -17655.065,E2 -17655.065} C_VEL
LIN {X 0,Y 270.292,Z 365.431,A -85,B 0,C 180,E1 -17659.756,E2 -17659.756} C_VEL
LIN {X 0,Y 270.264,Z 365.442,A -85,B 0,C 180,E1 -17664.586,E2 -17664.586} C_VEL
LIN {X 0,Y 270.235,Z 365.388,A -85,B 0,C 180,E1 -17667.913,E2 -17667.913} C_VEL
LIN {X 0,Y 270.164,Z 365.419,A -85,B 0,C 180,E1 -17671.351,E2 -17671.351} C_VEL
LIN {X 0,Y 270.206,Z 365.442,A -85,B 0,C 180,E1 -17674.905,E2 -17674.905} C_VEL
LIN {X 0,Y 270.214,Z 365.405,A -85,B 0,C 180,E1 -17678.718,E2 -17678.718} C_VEL
LIN {X 0,Y 270.256,Z 365.436,A -85,B 0,C 180,E1 -17682.542,E2 -17682.542} C_VEL
LIN {X 0,Y 270.229,Z 365.433,A -85,B 0,C 180,E1 -17686.737,E2 -17686.737} C_VEL
LIN {X 0,Y 270.296,Z 365.633,A -85,B 0,C 180,E1 -17689.818,E2 -17689.818} C_VEL
LIN {X 0,Y 272.129,Z 372.25,A -85,B 0,C 180,E1 -17692.504,E2 -17692.504} C_VEL
LIN {X 0,Y 279.414,Z 386.117,A -85,B 0,C 180,E1 -17694.128,E2 -17694.128} C_VEL
LIN {X 0,Y 286.816,Z 401.305,A -85,B 0,C 180,E1 -17695.643,E2 -17695.643} C_VEL
LIN {X 0,Y 293.399,Z 417.039,A -85,B 0,C 180,E1 -17696.97,E2 -17696.97} C_VEL
LIN {X 0,Y 293.941,Z 419.937,A -85,B 0,C 180,E1 -17697.121,E2 -17697.121} C_VEL
LIN {X 0,Y 291.277,Z 494.885,A -85,B 0,C 180,E1 -17698.92,E2 -17698.92} C_VEL
LIN {X 0,Y 290.464,Z 512.619,A -85,B 0,C 180,E1 -17699.415,E2 -17699.415} C_VEL
LIN {X 0,Y 289.125,Z 526.942,A -85,B 0,C 180,E1 -17700.064,E2 -17700.064} C_VEL
LIN {X 0,Y 287.276,Z 541.295,A -85,B 0,C 180,E1 -17701.01,E2 -17701.01} C_VEL
LIN {X 0,Y 285.212,Z 555.006,A -85,B 0,C 180,E1 -17702.26,E2 -17702.26} C_VEL
LIN {X 0,Y 283.066,Z 566.965,A -85,B 0,C 180,E1 -17703.656,E2 -17703.656} C_VEL
LIN {X 0,Y 280.494,Z 578.912,A -85,B 0,C 180,E1 -17705.385,E2 -17705.385} C_VEL
LIN {X 0,Y 277.975,Z 589.693,A -85,B 0,C 180,E1 -17707.323,E2 -17707.323} C_VEL
LIN {X 0,Y 275.555,Z 599.404,A -85,B 0,C 180,E1 -17709.473,E2 -17709.473} C_VEL
LIN {X 0,Y 273.524,Z 607.46,A -85,B 0,C 180,E1 -17711.656,E2 -17711.656} C_VEL
LIN {X 0,Y 271.806,Z 615.179,A -85,B 0,C 180,E1 -17714.249,E2 -17714.249} C_VEL
LIN {X 0,Y 270.368,Z 620.562,A -85,B 0,C 180,E1 -17716.472,E2 -17716.472} C_VEL
LIN {X 0,Y 269.193,Z 626.228,A -85,B 0,C 180,E1 -17719.472,E2 -17719.472} C_VEL
LIN {X 0,Y 268.48,Z 630.339,A -85,B 0,C 180,E1 -17722.481,E2 -17722.481} C_VEL
LIN {X 0,Y 268.171,Z 633.017,A -85,B 0,C 180,E1 -17725.493,E2 -17725.493} C_VEL
LIN {X 0,Y 268.128,Z 634.338,A -85,B 0,C 180,E1 -17728.5,E2 -17728.5} C_VEL
LIN {X 0,Y 268.128,Z 634.33,A -85,B 0,C 180,E1 -17731.504,E2 -17731.504} C_VEL
LIN {X 0,Y 268.16,Z 633.004,A -85,B 0,C 180,E1 -17734.511,E2 -17734.511} C_VEL
LIN {X 0,Y 268.625,Z 632.658,A -85,B 0,C 180,E1 -17737.518,E2 -17737.518} C_VEL
LIN {X 0,Y 268.964,Z 631.926,A -85,B 0,C 180,E1 -17739.022,E2 -17739.022} C_VEL
LIN {X 0,Y 269.513,Z 630.746,A -85,B 0,C 180,E1 -17740.519,E2 -17740.519} C_VEL
LIN {X 0,Y 270.975,Z 627.141,A -85,B 0,C 180,E1 -17743.501,E2 -17743.501} C_VEL
LIN {X 0,Y 272.56,Z 623.27,A -85,B 0,C 180,E1 -17745.71,E2 -17745.71} C_VEL
LIN {X 0,Y 274.913,Z 617.055,A -85,B 0,C 180,E1 -17748.391,E2 -17748.391} C_VEL
LIN {X 0,Y 277.55,Z 609.857,A -85,B 0,C 180,E1 -17750.765,E2 -17750.765} C_VEL
LIN {X 0,Y 280.341,Z 601.947,A -85,B 0,C 180,E1 -17752.868,E2 -17752.868} C_VEL
LIN {X 0,Y 283.481,Z 592.253,A -85,B 0,C 180,E1 -17754.929,E2 -17754.929} C_VEL
LIN {X 0,Y 286.794,Z 581.454,A -85,B 0,C 180,E1 -17756.764,E2 -17756.764} C_VEL
LIN {X 0,Y 290.255,Z 568.283,A -85,B 0,C 180,E1 -17758.57,E2 -17758.57} C_VEL
LIN {X 0,Y 293.218,Z 555.288,A -85,B 0,C 180,E1 -17759.942,E2 -17759.942} C_VEL
LIN {X 0,Y 295.751,Z 542.144,A -85,B 0,C 180,E1 -17761.024,E2 -17761.024} C_VEL
LIN {X 0,Y 298.141,Z 526.199,A -85,B 0,C 180,E1 -17761.98,E2 -17761.98} C_VEL
LIN {X 0,Y 302.841,Z 495.176,A -85,B 0,C 180,E1 -17763.399,E2 -17763.399} C_VEL
LIN {X 0,Y 313.444,Z 432.729,A -85,B 0,C 180,E1 -17766.117,E2 -17766.117} C_VEL
LIN {X 0,Y 310.352,Z 428.648,A -85,B 0,C 180,E1 -17768.391,E2 -17768.391} C_VEL
LIN {X 0,Y 308,Z 426.017,A -85,B 0,C 180,E1 -17770.859,E2 -17770.859} C_VEL
LIN {X 0,Y 306.798,Z 425.3,A -85,B 0,C 180,E1 -17772.858,E2 -17772.858} C_VEL
LIN {X 0,Y 306.169,Z 426.082,A -85,B 0,C 180,E1 -17775.367,E2 -17775.367} C_VEL
LIN {X 0,Y 306.502,Z 428.066,A -85,B 0,C 180,E1 -17777.642,E2 -17777.642} C_VEL
LIN {X 0,Y 307.663,Z 431.585,A -85,B 0,C 180,E1 -17779.931,E2 -17779.931} C_VEL
LIN {X 0,Y 309.577,Z 437.446,A -85,B 0,C 180,E1 -17782.282,E2 -17782.282} C_VEL
LIN {X 0,Y 310.661,Z 441.459,A -85,B 0,C 180,E1 -17783.411,E2 -17783.411} C_VEL
LIN {X 0,Y 311.058,Z 453.704,A -85,B 0,C 180,E1 -17785.04,E2 -17785.04} C_VEL
LIN {X 0,Y 311.25,Z 465.891,A -85,B 0,C 180,E1 -17786.366,E2 -17786.366} C_VEL
LIN {X 0,Y 311.12,Z 468.651,A -85,B 0,C 180,E1 -17786.589,E2 -17786.589} C_VEL
LIN {X 0,Y 301.209,Z 535.657,A -85,B 0,C 180,E1 -17789.504,E2 -17789.504} C_VEL
LIN {X 0,Y 298.475,Z 549.533,A -85,B 0,C 180,E1 -17790.365,E2 -17790.365} C_VEL
LIN {X 0,Y 295.105,Z 563.504,A -85,B 0,C 180,E1 -17791.556,E2 -17791.556} C_VEL
LIN {X 0,Y 291.958,Z 574.71,A -85,B 0,C 180,E1 -17792.783,E2 -17792.783} C_VEL
LIN {X 0,Y 288.424,Z 586.121,A -85,B 0,C 180,E1 -17794.369,E2 -17794.369} C_VEL
LIN {X 0,Y 285.169,Z 595.622,A -85,B 0,C 180,E1 -17796.005,E2 -17796.005} C_VEL
LIN {X 0,Y 281.524,Z 605.028,A -85,B 0,C 180,E1 -17798.009,E2 -17798.009} C_VEL
LIN {X 0,Y 278.423,Z 612.729,A -85,B 0,C 180,E1 -17800.076,E2 -17800.076} C_VEL
LIN {X 0,Y 275.651,Z 619.014,A -85,B 0,C 180,E1 -17802.185,E2 -17802.185} C_VEL
LIN {X 0,Y 273.575,Z 624.021,A -85,B 0,C 180,E1 -17804.351,E2 -17804.351} C_VEL
LIN {X 0,Y 271.815,Z 627.942,A -85,B 0,C 180,E1 -17806.544,E2 -17806.544} C_VEL
LIN {X 0,Y 269.951,Z 631.605,A -85,B 0,C 180,E1 -17809.5,E2 -17809.5} C_VEL
LIN {X 0,Y 269.292,Z 632.806,A -85,B 0,C 180,E1 -17810.991,E2 -17810.991} C_VEL
LIN {X 0,Y 268.827,Z 633.554,A -85,B 0,C 180,E1 -17812.489,E2 -17812.489} C_VEL
LIN {X 0,Y 268.405,Z 633.939,A -85,B 0,C 180,E1 -17814.283,E2 -17814.283} C_VEL
LIN {X 0,Y 268.171,Z 633.355,A -85,B 0,C 180,E1 -17816.996,E2 -17816.996} C_VEL
LIN {X 0,Y 268.161,Z 632.413,A -85,B 0,C 180,E1 -17818.498,E2 -17818.498} C_VEL
LIN {X 0,Y 268.133,Z 631.05,A -85,B 0,C 180,E1 -17820,E2 -17820} C_VEL
LIN {X 0,Y 268.205,Z 628.123,A -85,B 0,C 180,E1 -17822.253,E2 -17822.253} C_VEL
LIN {X 0,Y 268.313,Z 624.064,A -85,B 0,C 180,E1 -17824.507,E2 -17824.507} C_VEL
LIN {X 0,Y 268.489,Z 618.745,A -85,B 0,C 180,E1 -17826.765,E2 -17826.765} C_VEL
LIN {X 0,Y 268.883,Z 611.966,A -85,B 0,C 180,E1 -17829.023,E2 -17829.023} C_VEL
LIN {X 0,Y 269.444,Z 603.51,A -85,B 0,C 180,E1 -17831.281,E2 -17831.281} C_VEL
LIN {X 0,Y 270.104,Z 594.82,A -85,B 0,C 180,E1 -17833.16,E2 -17833.16} C_VEL
LIN {X 0,Y 271.06,Z 584.272,A -85,B 0,C 180,E1 -17835.027,E2 -17835.027} C_VEL
LIN {X 0,Y 271.903,Z 573.958,A -85,B 0,C 180,E1 -17836.518,E2 -17836.518} C_VEL
LIN {X 0,Y 272.912,Z 561.011,A -85,B 0,C 180,E1 -17838.001,E2 -17838.001} C_VEL
LIN {X 0,Y 273.697,Z 548.47,A -85,B 0,C 180,E1 -17839.111,E2 -17839.111} C_VEL
LIN {X 0,Y 274.53,Z 534.456,A -85,B 0,C 180,E1 -17840.023,E2 -17840.023} C_VEL
LIN {X 0,Y 275.56,Z 508.542,A -85,B 0,C 180,E1 -17841.116,E2 -17841.116} C_VEL
LIN {X 0,Y 277.541,Z 453.787,A -85,B 0,C 180,E1 -17843.296,E2 -17843.296} C_VEL
LIN {X 0,Y 275.061,Z 428.402,A -85,B 0,C 180,E1 -17844.431,E2 -17844.431} C_VEL
LIN {X 0,Y 274.601,Z 420.058,A -85,B 0,C 180,E1 -17844.828,E2 -17844.828} C_VEL
LIN {X 0,Y 276.314,Z 401.951,A -85,B 0,C 180,E1 -17848.484,E2 -17848.484} C_VEL
LIN {X 0,Y 276.91,Z 396.249,A -85,B 0,C 180,E1 -17849.639,E2 -17849.639} C_VEL
LIN {X 0,Y 274.758,Z 385.45,A -85,B 0,C 180,E1 -17852.04,E2 -17852.04} C_VEL
LIN {X 0,Y 270.561,Z 366.658,A -85,B 0,C 180,E1 -17856.364,E2 -17856.364} C_VEL
LIN {X 0,Y 270.291,Z 365.547,A -85,B 0,C 180,E1 -17856.73,E2 -17856.73} C_VEL
LIN {X 0,Y 270.175,Z 365.455,A -85,B 0,C 180,E1 -17861.027,E2 -17861.027} C_VEL
LIN {X 0,Y 270.158,Z 365.424,A -85,B 0,C 180,E1 -17865.379,E2 -17865.379} C_VEL
LIN {X 0,Y 270.222,Z 365.517,A -85,B 0,C 180,E1 -17869.799,E2 -17869.799} C_VEL
LIN {X 0,Y 271.714,Z 370.926,A -85,B 0,C 180,E1 -17872.136,E2 -17872.136} C_VEL
LIN {X 0,Y 272.218,Z 372.56,A -85,B 0,C 180,E1 -17872.651,E2 -17872.651} C_VEL
LIN {X 0,Y 280.861,Z 388.868,A -85,B 0,C 180,E1 -17874.512,E2 -17874.512} C_VEL
LIN {X 0,Y 289.252,Z 406.941,A -85,B 0,C 180,E1 -17876.22,E2 -17876.22} C_VEL
LIN {X 0,Y 293.529,Z 417.809,A -85,B 0,C 180,E1 -17877.088,E2 -17877.088} C_VEL
LIN {X 0,Y 293.951,Z 420.607,A -85,B 0,C 180,E1 -17877.221,E2 -17877.221} C_VEL
LIN {X 0,Y 290.577,Z 509.744,A -85,B 0,C 180,E1 -17879.38,E2 -17879.38} C_VEL
LIN {X 0,Y 289.344,Z 524.178,A -85,B 0,C 180,E1 -17879.984,E2 -17879.984} C_VEL
LIN {X 0,Y 287.665,Z 538.119,A -85,B 0,C 180,E1 -17880.848,E2 -17880.848} C_VEL
LIN {X 0,Y 285.778,Z 551.077,A -85,B 0,C 180,E1 -17881.942,E2 -17881.942} C_VEL
LIN {X 0,Y 283.598,Z 563.554,A -85,B 0,C 180,E1 -17883.296,E2 -17883.296} C_VEL
LIN {X 0,Y 281.28,Z 575.105,A -85,B 0,C 180,E1 -17884.863,E2 -17884.863} C_VEL
LIN {X 0,Y 278.865,Z 585.624,A -85,B 0,C 180,E1 -17886.612,E2 -17886.612} C_VEL
LIN {X 0,Y 276.387,Z 596.073,A -85,B 0,C 180,E1 -17888.754,E2 -17888.754} C_VEL
LIN {X 0,Y 274.166,Z 604.692,A -85,B 0,C 180,E1 -17890.921,E2 -17890.921} C_VEL
LIN {X 0,Y 272.639,Z 611.113,A -85,B 0,C 180,E1 -17892.884,E2 -17892.884} C_VEL
LIN {X 0,Y 271.326,Z 616.908,A -85,B 0,C 180,E1 -17894.986,E2 -17894.986} C_VEL
LIN {X 0,Y 270.016,Z 622.01,A -85,B 0,C 180,E1 -17897.216,E2 -17897.216} C_VEL
LIN {X 0,Y 268.977,Z 627.294,A -85,B 0,C 180,E1 -17900.22,E2 -17900.22} C_VEL
LIN {X 0,Y 268.483,Z 630.243,A -85,B 0,C 180,E1 -17902.478,E2 -17902.478} C_VEL
LIN {X 0,Y 268.162,Z 632.957,A -85,B 0,C 180,E1 -17905.489,E2 -17905.489} C_VEL
LIN {X 0,Y 268.129,Z 634.317,A -85,B 0,C 180,E1 -17908.496,E2 -17908.496} C_VEL
LIN {X 0,Y 268.129,Z 634.348,A -85,B 0,C 180,E1 -17911.5,E2 -17911.5} C_VEL
LIN {X 0,Y 268.162,Z 633.051,A -85,B 0,C 180,E1 -17914.508,E2 -17914.508} C_VEL
LIN {X 0,Y 268.481,Z 630.392,A -85,B 0,C 180,E1 -17917.519,E2 -17917.519} C_VEL
LIN {X 0,Y 269.19,Z 626.302,A -85,B 0,C 180,E1 -17920.528,E2 -17920.528} C_VEL
LIN {X 0,Y 270.357,Z 620.656,A -85,B 0,C 180,E1 -17923.528,E2 -17923.528} C_VEL
LIN {X 0,Y 271.92,Z 614.289,A -85,B 0,C 180,E1 -17926.129,E2 -17926.129} C_VEL
LIN {X 0,Y 273.827,Z 606.372,A -85,B 0,C 180,E1 -17928.711,E2 -17928.711} C_VEL
LIN {X 0,Y 275.897,Z 598.091,A -85,B 0,C 180,E1 -17930.891,E2 -17930.891} C_VEL
LIN {X 0,Y 278.318,Z 588.116,A -85,B 0,C 180,E1 -17933.04,E2 -17933.04} C_VEL
LIN {X 0,Y 280.934,Z 577.011,A -85,B 0,C 180,E1 -17934.968,E2 -17934.968} C_VEL
LIN {X 0,Y 283.232,Z 565.961,A -85,B 0,C 180,E1 -17936.526,E2 -17936.526} C_VEL
LIN {X 0,Y 285.406,Z 553.959,A -85,B 0,C 180,E1 -17937.894,E2 -17937.894} C_VEL
LIN {X 0,Y 287.388,Z 540.673,A -85,B 0,C 180,E1 -17939.078,E2 -17939.078} C_VEL
LIN {X 0,Y 289.093,Z 526.862,A -85,B 0,C 180,E1 -17939.99,E2 -17939.99} C_VEL
LIN {X 0,Y 290.465,Z 512.472,A -85,B 0,C 180,E1 -17940.636,E2 -17940.636} C_VEL
LIN {X 0,Y 291.405,Z 492.37,A -85,B 0,C 180,E1 -17941.181,E2 -17941.181} C_VEL
LIN {X 0,Y 293.898,Z 419.759,A -85,B 0,C 180,E1 -17942.935,E2 -17942.935} C_VEL
LIN {X 0,Y 292.874,Z 415.682,A -85,B 0,C 180,E1 -17943.181,E2 -17943.181} C_VEL
LIN {X 0,Y 286.809,Z 401.377,A -85,B 0,C 180,E1 -17944.4,E2 -17944.4} C_VEL
LIN {X 0,Y 280.326,Z 387.951,A -85,B 0,C 180,E1 -17945.726,E2 -17945.726} C_VEL
LIN {X 0,Y 273.725,Z 375.457,A -85,B 0,C 180,E1 -17947.127,E2 -17947.127} C_VEL
LIN {X 0,Y 273.586,Z 375.224,A -85,B 0,C 180,E1 -17947.156,E2 -17947.156} C_VEL
LIN {X 0,Y 271.954,Z 373.157,A -85,B 0,C 180,E1 -17947.534,E2 -17947.534} C_VEL
LIN {X 0,Y 269.225,Z 371.526,A -85,B 0,C 180,E1 -17948.235,E2 -17948.235} C_VEL
LIN {X 0,Y 264.97,Z 369.45,A -85,B 0,C 180,E1 -17949.703,E2 -17949.703} C_VEL
LIN {X 0,Y 263.675,Z 367.948,A -85,B 0,C 180,E1 -17950.511,E2 -17950.511} C_VEL
LIN {X 0,Y 263.455,Z 367.356,A -85,B 0,C 180,E1 -17950.785,E2 -17950.785} C_VEL
LIN {X 0,Y 263.213,Z 366.339,A -85,B 0,C 180,E1 -17951.412,E2 -17951.412} C_VEL
LIN {X 0,Y 263.186,Z 366.298,A -85,B 0,C 180,E1 -17953.968,E2 -17953.968} C_VEL
LIN {X 0,Y 263.209,Z 366.325,A -85,B 0,C 180,E1 -17958.382,E2 -17958.382} C_VEL
LIN {X 0,Y 263.197,Z 366.279,A -85,B 0,C 180,E1 -17963.229,E2 -17963.229} C_VEL
LIN {X 0,Y 263.176,Z 366.328,A -85,B 0,C 180,E1 -17965.889,E2 -17965.889} C_VEL
LIN {X 0,Y 263.132,Z 366.278,A -85,B 0,C 180,E1 -17969.504,E2 -17969.504} C_VEL
LIN {X 0,Y 263.184,Z 366.279,A -85,B 0,C 180,E1 -17973.002,E2 -17973.002} C_VEL
LIN {X 0,Y 263.182,Z 366.327,A -85,B 0,C 180,E1 -17976.387,E2 -17976.387} C_VEL
LIN {X 0,Y 263.254,Z 366.302,A -85,B 0,C 180,E1 -17979.692,E2 -17979.692} C_VEL
LIN {X 0,Y 263.341,Z 366.283,A -85,B 0,C 180,E1 -17984.521,E2 -17984.521} C_VEL
LIN {X 0,Y 263.365,Z 366.286,A -85,B 0,C 180,E1 -17989.234,E2 -17989.234} C_VEL
LIN {X 0,Y 263.563,Z 366.271,A -85,B 0,C 180,E1 -17992.338,E2 -17992.338} C_VEL
LIN {X 0,Y 263.744,Z 366.248,A -85,B 0,C 180,E1 -17998.473,E2 -17998.473} C_VEL
LIN {X 0,Y 263.744,Z 366.248,A -85,B 0,C 180,E1 -18001.527,E2 -18001.527} C_VEL
LIN {X 0,Y 263.563,Z 366.272,A -85,B 0,C 180,E1 -18007.662,E2 -18007.662} C_VEL
LIN {X 0,Y 263.364,Z 366.285,A -85,B 0,C 180,E1 -18010.766,E2 -18010.766} C_VEL
LIN {X 0,Y 263.341,Z 366.281,A -85,B 0,C 180,E1 -18015.479,E2 -18015.479} C_VEL
LIN {X 0,Y 263.254,Z 366.301,A -85,B 0,C 180,E1 -18020.307,E2 -18020.307} C_VEL
LIN {X 0,Y 263.197,Z 366.315,A -85,B 0,C 180,E1 -18025.292,E2 -18025.292} C_VEL
LIN {X 0,Y 263.145,Z 366.264,A -85,B 0,C 180,E1 -18028.734,E2 -18028.734} C_VEL
LIN {X 0,Y 263.12,Z 366.318,A -85,B 0,C 180,E1 -18032.29,E2 -18032.29} C_VEL
LIN {X 0,Y 263.18,Z 366.293,A -85,B 0,C 180,E1 -18035.979,E2 -18035.979} C_VEL
LIN {X 0,Y 263.155,Z 366.3,A -85,B 0,C 180,E1 -18039.863,E2 -18039.863} C_VEL
LIN {X 0,Y 263.206,Z 366.324,A -85,B 0,C 180,E1 -18041.877,E2 -18041.877} C_VEL
LIN {X 0,Y 263.185,Z 366.299,A -85,B 0,C 180,E1 -18046.137,E2 -18046.137} C_VEL
LIN {X 0,Y 263.211,Z 366.358,A -85,B 0,C 180,E1 -18048.7,E2 -18048.7} C_VEL
LIN {X 0,Y 264.263,Z 370.112,A -85,B 0,C 180,E1 -18050.466,E2 -18050.466} C_VEL
LIN {X 0,Y 264.895,Z 372.393,A -85,B 0,C 180,E1 -18051.316,E2 -18051.316} C_VEL
LIN {X 0,Y 272.055,Z 385.494,A -85,B 0,C 180,E1 -18052.978,E2 -18052.978} C_VEL
LIN {X 0,Y 279.619,Z 400.798,A -85,B 0,C 180,E1 -18054.613,E2 -18054.613} C_VEL
LIN {X 0,Y 286.147,Z 415.752,A -85,B 0,C 180,E1 -18055.981,E2 -18055.981} C_VEL
LIN {X 0,Y 287.851,Z 420.403,A -85,B 0,C 180,E1 -18056.347,E2 -18056.347} C_VEL
LIN {X 0,Y 287.767,Z 428.5,A -85,B 0,C 180,E1 -18056.573,E2 -18056.573} C_VEL
LIN {X 0,Y 284.61,Z 509.444,A -85,B 0,C 180,E1 -18058.571,E2 -18058.571} C_VEL
LIN {X 0,Y 283.357,Z 523.904,A -85,B 0,C 180,E1 -18059.183,E2 -18059.183} C_VEL
LIN {X 0,Y 281.588,Z 537.913,A -85,B 0,C 180,E1 -18060.057,E2 -18060.057} C_VEL
LIN {X 0,Y 279.797,Z 550.041,A -85,B 0,C 180,E1 -18061.086,E2 -18061.086} C_VEL
LIN {X 0,Y 277.439,Z 563.074,A -85,B 0,C 180,E1 -18062.504,E2 -18062.504} C_VEL
LIN {X 0,Y 274.878,Z 575.59,A -85,B 0,C 180,E1 -18064.239,E2 -18064.239} C_VEL
LIN {X 0,Y 272.287,Z 586.028,A -85,B 0,C 180,E1 -18066.016,E2 -18066.016} C_VEL
LIN {X 0,Y 269.715,Z 596.409,A -85,B 0,C 180,E1 -18068.206,E2 -18068.206} C_VEL
LIN {X 0,Y 267.397,Z 604.972,A -85,B 0,C 180,E1 -18070.423,E2 -18070.423} C_VEL
LIN {X 0,Y 265.357,Z 613.166,A -85,B 0,C 180,E1 -18073.064,E2 -18073.064} C_VEL
LIN {X 0,Y 263.943,Z 618.903,A -85,B 0,C 180,E1 -18075.35,E2 -18075.35} C_VEL
LIN {X 0,Y 262.704,Z 623.6,A -85,B 0,C 180,E1 -18077.644,E2 -18077.644} C_VEL
LIN {X 0,Y 261.738,Z 628.47,A -85,B 0,C 180,E1 -18080.731,E2 -18080.731} C_VEL
LIN {X 0,Y 261.231,Z 631.852,A -85,B 0,C 180,E1 -18083.824,E2 -18083.824} C_VEL
LIN {X 0,Y 261.018,Z 633.845,A -85,B 0,C 180,E1 -18086.915,E2 -18086.915} C_VEL
LIN {X 0,Y 261.035,Z 634.5,A -85,B 0,C 180,E1 -18090.002,E2 -18090.002} C_VEL
LIN {X 0,Y 261.017,Z 633.827,A -85,B 0,C 180,E1 -18093.089,E2 -18093.089} C_VEL
LIN {X 0,Y 261.117,Z 632.965,A -85,B 0,C 180,E1 -18095.215,E2 -18095.215} C_VEL
LIN {X 0,Y 261.568,Z 632.837,A -85,B 0,C 180,E1 -18097.723,E2 -18097.723} C_VEL
LIN {X 0,Y 262.535,Z 631.195,A -85,B 0,C 180,E1 -18100.802,E2 -18100.802} C_VEL
LIN {X 0,Y 263.243,Z 629.775,A -85,B 0,C 180,E1 -18102.334,E2 -18102.334} C_VEL
LIN {X 0,Y 264.664,Z 626.814,A -85,B 0,C 180,E1 -18104.614,E2 -18104.614} C_VEL
LIN {X 0,Y 266.449,Z 622.884,A -85,B 0,C 180,E1 -18106.868,E2 -18106.868} C_VEL
LIN {X 0,Y 268.581,Z 617.864,A -85,B 0,C 180,E1 -18109.094,E2 -18109.094} C_VEL
LIN {X 0,Y 271.625,Z 610.506,A -85,B 0,C 180,E1 -18111.637,E2 -18111.637} C_VEL
LIN {X 0,Y 275.154,Z 601.339,A -85,B 0,C 180,E1 -18114.123,E2 -18114.123} C_VEL
LIN {X 0,Y 278.685,Z 591.582,A -85,B 0,C 180,E1 -18116.19,E2 -18116.19} C_VEL
LIN {X 0,Y 282.281,Z 580.77,A -85,B 0,C 180,E1 -18118.032,E2 -18118.032} C_VEL
LIN {X 0,Y 285.929,Z 568.084,A -85,B 0,C 180,E1 -18119.78,E2 -18119.78} C_VEL
LIN {X 0,Y 289.095,Z 555.545,A -85,B 0,C 180,E1 -18121.106,E2 -18121.106} C_VEL
LIN {X 0,Y 291.873,Z 542.577,A -85,B 0,C 180,E1 -18122.193,E2 -18122.193} C_VEL
LIN {X 0,Y 294.347,Z 527.779,A -85,B 0,C 180,E1 -18123.107,E2 -18123.107} C_VEL
LIN {X 0,Y 299.53,Z 496.122,A -85,B 0,C 180,E1 -18124.579,E2 -18124.579} C_VEL
LIN {X 0,Y 310.075,Z 437.755,A -85,B 0,C 180,E1 -18127.141,E2 -18127.141} C_VEL
LIN {X 0,Y 307.637,Z 434.573,A -85,B 0,C 180,E1 -18129.21,E2 -18129.21} C_VEL
LIN {X 0,Y 305.944,Z 432.641,A -85,B 0,C 180,E1 -18131.297,E2 -18131.297} C_VEL
LIN {X 0,Y 305.209,Z 432.247,A -85,B 0,C 180,E1 -18132.536,E2 -18132.536} C_VEL
LIN {X 0,Y 304.456,Z 432.749,A -85,B 0,C 180,E1 -18134.994,E2 -18134.994} C_VEL
LIN {X 0,Y 304.629,Z 434.711,A -85,B 0,C 180,E1 -18137.335,E2 -18137.335} C_VEL
LIN {X 0,Y 305.563,Z 438.04,A -85,B 0,C 180,E1 -18139.531,E2 -18139.531} C_VEL
LIN {X 0,Y 307.084,Z 443.45,A -85,B 0,C 180,E1 -18141.749,E2 -18141.749} C_VEL
LIN {X 0,Y 307.785,Z 446.645,A -85,B 0,C 180,E1 -18142.643,E2 -18142.643} C_VEL
LIN {X 0,Y 307.806,Z 459.032,A -85,B 0,C 180,E1 -18144.293,E2 -18144.293} C_VEL
LIN {X 0,Y 307.684,Z 469.846,A -85,B 0,C 180,E1 -18145.461,E2 -18145.461} C_VEL
LIN {X 0,Y 297.208,Z 535.772,A -85,B 0,C 180,E1 -18148.373,E2 -18148.373} C_VEL
LIN {X 0,Y 294.297,Z 549.605,A -85,B 0,C 180,E1 -18149.247,E2 -18149.247} C_VEL
LIN {X 0,Y 290.576,Z 563.964,A -85,B 0,C 180,E1 -18150.475,E2 -18150.475} C_VEL
LIN {X 0,Y 286.835,Z 576.197,A -85,B 0,C 180,E1 -18151.858,E2 -18151.858} C_VEL
LIN {X 0,Y 283.091,Z 587.294,A -85,B 0,C 180,E1 -18153.457,E2 -18153.457} C_VEL
LIN {X 0,Y 279.466,Z 596.922,A -85,B 0,C 180,E1 -18155.194,E2 -18155.194} C_VEL
LIN {X 0,Y 275.77,Z 605.697,A -85,B 0,C 180,E1 -18157.13,E2 -18157.13} C_VEL
LIN {X 0,Y 272.466,Z 613.212,A -85,B 0,C 180,E1 -18159.227,E2 -18159.227} C_VEL
LIN {X 0,Y 269.028,Z 620.266,A -85,B 0,C 180,E1 -18161.731,E2 -18161.731} C_VEL
LIN {X 0,Y 266.819,Z 624.99,A -85,B 0,C 180,E1 -18163.945,E2 -18163.945} C_VEL
LIN {X 0,Y 264.955,Z 628.655,A -85,B 0,C 180,E1 -18166.189,E2 -18166.189} C_VEL
LIN {X 0,Y 263.898,Z 630.566,A -85,B 0,C 180,E1 -18167.699,E2 -18167.699} C_VEL
LIN {X 0,Y 262.997,Z 632.022,A -85,B 0,C 180,E1 -18169.219,E2 -18169.219} C_VEL
LIN {X 0,Y 261.784,Z 633.698,A -85,B 0,C 180,E1 -18172.286,E2 -18172.286} C_VEL
LIN {X 0,Y 261.299,Z 633.886,A -85,B 0,C 180,E1 -18174.378,E2 -18174.378} C_VEL
LIN {X 0,Y 261.091,Z 633.086,A -85,B 0,C 180,E1 -18176.914,E2 -18176.914} C_VEL
LIN {X 0,Y 261.091,Z 632.048,A -85,B 0,C 180,E1 -18178.458,E2 -18178.458} C_VEL
LIN {X 0,Y 261.062,Z 630.556,A -85,B 0,C 180,E1 -18180,E2 -18180} C_VEL
LIN {X 0,Y 261.143,Z 627.424,A -85,B 0,C 180,E1 -18182.314,E2 -18182.314} C_VEL
LIN {X 0,Y 261.273,Z 623.139,A -85,B 0,C 180,E1 -18184.629,E2 -18184.629} C_VEL
LIN {X 0,Y 261.45,Z 617.559,A -85,B 0,C 180,E1 -18186.948,E2 -18186.948} C_VEL
LIN {X 0,Y 261.881,Z 610.535,A -85,B 0,C 180,E1 -18189.266,E2 -18189.266} C_VEL
LIN {X 0,Y 262.438,Z 601.692,A -85,B 0,C 180,E1 -18191.587,E2 -18191.587} C_VEL
LIN {X 0,Y 263.263,Z 591.7,A -85,B 0,C 180,E1 -18193.705,E2 -18193.705} C_VEL
LIN {X 0,Y 264.237,Z 580.366,A -85,B 0,C 180,E1 -18195.623,E2 -18195.623} C_VEL
LIN {X 0,Y 265.16,Z 569.448,A -85,B 0,C 180,E1 -18197.118,E2 -18197.118} C_VEL
LIN {X 0,Y 266.107,Z 556.876,A -85,B 0,C 180,E1 -18198.477,E2 -18198.477} C_VEL
LIN {X 0,Y 266.908,Z 544.503,A -85,B 0,C 180,E1 -18199.517,E2 -18199.517} C_VEL
LIN {X 0,Y 267.763,Z 529.655,A -85,B 0,C 180,E1 -18200.402,E2 -18200.402} C_VEL
LIN {X 0,Y 270.553,Z 454.471,A -85,B 0,C 180,E1 -18203.526,E2 -18203.526} C_VEL
LIN {X 0,Y 268.109,Z 428.7,A -85,B 0,C 180,E1 -18204.718,E2 -18204.718} C_VEL
LIN {X 0,Y 267.629,Z 419.914,A -85,B 0,C 180,E1 -18205.156,E2 -18205.156} C_VEL
LIN {X 0,Y 269.411,Z 401.946,A -85,B 0,C 180,E1 -18208.856,E2 -18208.856} C_VEL
LIN {X 0,Y 269.905,Z 396.726,A -85,B 0,C 180,E1 -18209.937,E2 -18209.937} C_VEL
LIN {X 0,Y 266.407,Z 380.524,A -85,B 0,C 180,E1 -18213.642,E2 -18213.642} C_VEL
LIN {X 0,Y 263.248,Z 366.535,A -85,B 0,C 180,E1 -18216.995,E2 -18216.995} C_VEL
LIN {X 0,Y 263.13,Z 366.334,A -85,B 0,C 180,E1 -18221.593,E2 -18221.593} C_VEL
LIN {X 0,Y 263.111,Z 366.308,A -85,B 0,C 180,E1 -18226.154,E2 -18226.154} C_VEL
LIN {X 0,Y 263.182,Z 366.547,A -85,B 0,C 180,E1 -18228.958,E2 -18228.958} C_VEL
LIN {X 0,Y 264.834,Z 372.211,A -85,B 0,C 180,E1 -18231.37,E2 -18231.37} C_VEL
LIN {X 0,Y 269.262,Z 380.348,A -85,B 0,C 180,E1 -18232.45,E2 -18232.45} C_VEL
LIN {X 0,Y 277.437,Z 396.157,A -85,B 0,C 180,E1 -18234.234,E2 -18234.234} C_VEL
LIN {X 0,Y 284.528,Z 411.883,A -85,B 0,C 180,E1 -18235.729,E2 -18235.729} C_VEL
LIN {X 0,Y 287.831,Z 420.62,A -85,B 0,C 180,E1 -18236.433,E2 -18236.433} C_VEL
LIN {X 0,Y 285.531,Z 485.835,A -85,B 0,C 180,E1 -18238.04,E2 -18238.04} C_VEL
LIN {X 0,Y 284.426,Z 510.858,A -85,B 0,C 180,E1 -18238.694,E2 -18238.694} C_VEL
LIN {X 0,Y 283.145,Z 524.95,A -85,B 0,C 180,E1 -18239.309,E2 -18239.309} C_VEL
LIN {X 0,Y 281.494,Z 538.126,A -85,B 0,C 180,E1 -18240.145,E2 -18240.145} C_VEL
LIN {X 0,Y 279.527,Z 551.083,A -85,B 0,C 180,E1 -18241.257,E2 -18241.257} C_VEL
LIN {X 0,Y 277.299,Z 563.248,A -85,B 0,C 180,E1 -18242.594,E2 -18242.594} C_VEL
LIN {X 0,Y 274.863,Z 575.109,A -85,B 0,C 180,E1 -18244.234,E2 -18244.234} C_VEL
LIN {X 0,Y 272.327,Z 585.627,A -85,B 0,C 180,E1 -18246.015,E2 -18246.015} C_VEL
LIN {X 0,Y 269.739,Z 596.075,A -85,B 0,C 180,E1 -18248.204,E2 -18248.204} C_VEL
LIN {X 0,Y 267.447,Z 604.694,A -85,B 0,C 180,E1 -18250.423,E2 -18250.423} C_VEL
LIN {X 0,Y 265.362,Z 612.956,A -85,B 0,C 180,E1 -18253.061,E2 -18253.061} C_VEL
LIN {X 0,Y 263.953,Z 618.719,A -85,B 0,C 180,E1 -18255.346,E2 -18255.346} C_VEL
LIN {X 0,Y 262.724,Z 623.455,A -85,B 0,C 180,E1 -18257.641,E2 -18257.641} C_VEL
LIN {X 0,Y 261.743,Z 628.358,A -85,B 0,C 180,E1 -18260.727,E2 -18260.727} C_VEL
LIN {X 0,Y 261.231,Z 631.773,A -85,B 0,C 180,E1 -18263.82,E2 -18263.82} C_VEL
LIN {X 0,Y 261.018,Z 633.803,A -85,B 0,C 180,E1 -18266.911,E2 -18266.911} C_VEL
LIN {X 0,Y 261.036,Z 634.498,A -85,B 0,C 180,E1 -18269.998,E2 -18269.998} C_VEL
LIN {X 0,Y 261.017,Z 633.866,A -85,B 0,C 180,E1 -18273.085,E2 -18273.085} C_VEL
LIN {X 0,Y 261.229,Z 631.894,A -85,B 0,C 180,E1 -18276.176,E2 -18276.176} C_VEL
LIN {X 0,Y 261.739,Z 628.532,A -85,B 0,C 180,E1 -18279.269,E2 -18279.269} C_VEL
LIN {X 0,Y 262.695,Z 623.681,A -85,B 0,C 180,E1 -18282.356,E2 -18282.356} C_VEL
LIN {X 0,Y 264.414,Z 617.198,A -85,B 0,C 180,E1 -18285.412,E2 -18285.412} C_VEL
LIN {X 0,Y 266.129,Z 610.007,A -85,B 0,C 180,E1 -18288.066,E2 -18288.066} C_VEL
LIN {X 0,Y 268.464,Z 601.052,A -85,B 0,C 180,E1 -18290.694,E2 -18290.694} C_VEL
LIN {X 0,Y 270.893,Z 591.675,A -85,B 0,C 180,E1 -18292.9,E2 -18292.9} C_VEL
LIN {X 0,Y 273.475,Z 581.29,A -85,B 0,C 180,E1 -18294.884,E2 -18294.884} C_VEL
LIN {X 0,Y 276.108,Z 569.835,A -85,B 0,C 180,E1 -18296.653,E2 -18296.653} C_VEL
LIN {X 0,Y 278.276,Z 558.724,A -85,B 0,C 180,E1 -18298.056,E2 -18298.056} C_VEL
LIN {X 0,Y 280.327,Z 546.76,A -85,B 0,C 180,E1 -18299.265,E2 -18299.265} C_VEL
LIN {X 0,Y 282.071,Z 534.959,A -85,B 0,C 180,E1 -18300.195,E2 -18300.195} C_VEL
LIN {X 0,Y 283.599,Z 521.343,A -85,B 0,C 180,E1 -18300.994,E2 -18300.994} C_VEL
LIN {X 0,Y 284.692,Z 507.823,A -85,B 0,C 180,E1 -18301.524,E2 -18301.524} C_VEL
LIN {X 0,Y 287.996,Z 422.18,A -85,B 0,C 180,E1 -18303.627,E2 -18303.627} C_VEL
LIN {X 0,Y 287.339,Z 418.774,A -85,B 0,C 180,E1 -18303.814,E2 -18303.814} C_VEL
LIN {X 0,Y 281.198,Z 404.244,A -85,B 0,C 180,E1 -18305.099,E2 -18305.099} C_VEL
LIN {X 0,Y 275.05,Z 391.467,A -85,B 0,C 180,E1 -18306.408,E2 -18306.408} C_VEL
LIN {X 0,Y 268.464,Z 378.917,A -85,B 0,C 180,E1 -18307.866,E2 -18307.866} C_VEL
LIN {X 0,Y 264.814,Z 372.191,A -85,B 0,C 180,E1 -18308.776,E2 -18308.776} C_VEL
LIN {X 0,Y 263.455,Z 367.356,A -85,B 0,C 180,E1 -18310.785,E2 -18310.785} C_VEL
LIN {X 0,Y 262.775,Z 366.496,A -85,B 0,C 180,E1 -18311.571,E2 -18311.571} C_VEL
LIN {X 0,Y 259.31,Z 366.779,A -85,B 0,C 180,E1 -18314.045,E2 -18314.045} C_VEL
LIN {X 0,Y 257.081,Z 367.171,A -85,B 0,C 180,E1 -18315.779,E2 -18315.779} C_VEL
LIN {X 0,Y 256.146,Z 367.192,A -85,B 0,C 180,E1 -18317.575,E2 -18317.575} C_VEL
LIN {X 0,Y 256.102,Z 367.166,A -85,B 0,C 180,E1 -18320.863,E2 -18320.863} C_VEL
LIN {X 0,Y 256.113,Z 367.188,A -85,B 0,C 180,E1 -18324.812,E2 -18324.812} C_VEL
LIN {X 0,Y 256.084,Z 367.172,A -85,B 0,C 180,E1 -18328.571,E2 -18328.571} C_VEL
LIN {X 0,Y 256.13,Z 367.144,A -85,B 0,C 180,E1 -18332.195,E2 -18332.195} C_VEL
LIN {X 0,Y 256.164,Z 367.202,A -85,B 0,C 180,E1 -18335.699,E2 -18335.699} C_VEL
LIN {X 0,Y 256.157,Z 367.182,A -85,B 0,C 180,E1 -18339.104,E2 -18339.104} C_VEL
LIN {X 0,Y 256.29,Z 367.162,A -85,B 0,C 180,E1 -18344.084,E2 -18344.084} C_VEL
LIN {X 0,Y 256.3,Z 367.169,A -85,B 0,C 180,E1 -18348.933,E2 -18348.933} C_VEL
LIN {X 0,Y 256.53,Z 367.142,A -85,B 0,C 180,E1 -18352.127,E2 -18352.127} C_VEL
LIN {X 0,Y 256.706,Z 367.123,A -85,B 0,C 180,E1 -18358.431,E2 -18358.431} C_VEL
LIN {X 0,Y 256.706,Z 367.124,A -85,B 0,C 180,E1 -18361.569,E2 -18361.569} C_VEL
LIN {X 0,Y 256.53,Z 367.143,A -85,B 0,C 180,E1 -18367.873,E2 -18367.873} C_VEL
LIN {X 0,Y 256.3,Z 367.167,A -85,B 0,C 180,E1 -18371.066,E2 -18371.066} C_VEL
LIN {X 0,Y 256.29,Z 367.16,A -85,B 0,C 180,E1 -18375.915,E2 -18375.915} C_VEL
LIN {X 0,Y 256.157,Z 367.181,A -85,B 0,C 180,E1 -18380.896,E2 -18380.896} C_VEL
LIN {X 0,Y 256.178,Z 367.192,A -85,B 0,C 180,E1 -18385.139,E2 -18385.139} C_VEL
LIN {X 0,Y 256.104,Z 367.14,A -85,B 0,C 180,E1 -18388.586,E2 -18388.586} C_VEL
LIN {X 0,Y 256.075,Z 367.213,A -85,B 0,C 180,E1 -18393.292,E2 -18393.292} C_VEL
LIN {X 0,Y 256.131,Z 367.154,A -85,B 0,C 180,E1 -18397.28,E2 -18397.28} C_VEL
LIN {X 0,Y 256.128,Z 367.204,A -85,B 0,C 180,E1 -18401.189,E2 -18401.189} C_VEL
LIN {X 0,Y 256.111,Z 367.173,A -85,B 0,C 180,E1 -18405.518,E2 -18405.518} C_VEL
LIN {X 0,Y 256.161,Z 367.374,A -85,B 0,C 180,E1 -18407.797,E2 -18407.797} C_VEL
LIN {X 0,Y 257.66,Z 372.38,A -85,B 0,C 180,E1 -18410.011,E2 -18410.011} C_VEL
LIN {X 0,Y 265.742,Z 386.916,A -85,B 0,C 180,E1 -18411.991,E2 -18411.991} C_VEL
LIN {X 0,Y 274.193,Z 403.887,A -85,B 0,C 180,E1 -18413.901,E2 -18413.901} C_VEL
LIN {X 0,Y 280.943,Z 419.577,A -85,B 0,C 180,E1 -18415.378,E2 -18415.378} C_VEL
LIN {X 0,Y 282.062,Z 422.471,A -85,B 0,C 180,E1 -18415.622,E2 -18415.622} C_VEL
LIN {X 0,Y 279.098,Z 498.189,A -85,B 0,C 180,E1 -18417.498,E2 -18417.498} C_VEL
LIN {X 0,Y 278.288,Z 513.759,A -85,B 0,C 180,E1 -18417.974,E2 -18417.974} C_VEL
LIN {X 0,Y 276.837,Z 527.721,A -85,B 0,C 180,E1 -18418.641,E2 -18418.641} C_VEL
LIN {X 0,Y 274.955,Z 541.308,A -85,B 0,C 180,E1 -18419.577,E2 -18419.577} C_VEL
LIN {X 0,Y 272.993,Z 553.58,A -85,B 0,C 180,E1 -18420.718,E2 -18420.718} C_VEL
LIN {X 0,Y 270.638,Z 565.661,A -85,B 0,C 180,E1 -18422.135,E2 -18422.135} C_VEL
LIN {X 0,Y 267.96,Z 577.849,A -85,B 0,C 180,E1 -18423.942,E2 -18423.942} C_VEL
LIN {X 0,Y 265.329,Z 587.917,A -85,B 0,C 180,E1 -18425.762,E2 -18425.762} C_VEL
LIN {X 0,Y 262.69,Z 597.924,A -85,B 0,C 180,E1 -18428.005,E2 -18428.005} C_VEL
LIN {X 0,Y 260.319,Z 606.233,A -85,B 0,C 180,E1 -18430.279,E2 -18430.279} C_VEL
LIN {X 0,Y 258.254,Z 614.175,A -85,B 0,C 180,E1 -18432.992,E2 -18432.992} C_VEL
LIN {X 0,Y 257.046,Z 618.904,A -85,B 0,C 180,E1 -18434.947,E2 -18434.947} C_VEL
LIN {X 0,Y 255.728,Z 623.601,A -85,B 0,C 180,E1 -18437.301,E2 -18437.301} C_VEL
LIN {X 0,Y 254.724,Z 628.471,A -85,B 0,C 180,E1 -18440.473,E2 -18440.473} C_VEL
LIN {X 0,Y 254.159,Z 631.852,A -85,B 0,C 180,E1 -18443.652,E2 -18443.652} C_VEL
LIN {X 0,Y 253.923,Z 633.846,A -85,B 0,C 180,E1 -18446.829,E2 -18446.829} C_VEL
LIN {X 0,Y 253.944,Z 634.5,A -85,B 0,C 180,E1 -18450.002,E2 -18450.002} C_VEL
LIN {X 0,Y 253.92,Z 633.826,A -85,B 0,C 180,E1 -18453.175,E2 -18453.175} C_VEL
LIN {X 0,Y 254.022,Z 632.819,A -85,B 0,C 180,E1 -18455.121,E2 -18455.121} C_VEL
LIN {X 0,Y 254.517,Z 632.978,A -85,B 0,C 180,E1 -18457.938,E2 -18457.938} C_VEL
LIN {X 0,Y 254.932,Z 632.513,A -85,B 0,C 180,E1 -18459.523,E2 -18459.523} C_VEL
LIN {X 0,Y 256.312,Z 630.328,A -85,B 0,C 180,E1 -18462.673,E2 -18462.673} C_VEL
LIN {X 0,Y 257.864,Z 627.631,A -85,B 0,C 180,E1 -18465.008,E2 -18465.008} C_VEL
LIN {X 0,Y 260.464,Z 622.545,A -85,B 0,C 180,E1 -18468.079,E2 -18468.079} C_VEL
LIN {X 0,Y 263.362,Z 616.457,A -85,B 0,C 180,E1 -18470.726,E2 -18470.726} C_VEL
LIN {X 0,Y 266.852,Z 608.902,A -85,B 0,C 180,E1 -18473.271,E2 -18473.271} C_VEL
LIN {X 0,Y 270.209,Z 600.872,A -85,B 0,C 180,E1 -18475.416,E2 -18475.416} C_VEL
LIN {X 0,Y 274.113,Z 591.104,A -85,B 0,C 180,E1 -18477.486,E2 -18477.486} C_VEL
LIN {X 0,Y 277.968,Z 580.356,A -85,B 0,C 180,E1 -18479.334,E2 -18479.334} C_VEL
LIN {X 0,Y 282.086,Z 567.232,A -85,B 0,C 180,E1 -18481.131,E2 -18481.131} C_VEL
LIN {X 0,Y 285.632,Z 554.474,A -85,B 0,C 180,E1 -18482.454,E2 -18482.454} C_VEL
LIN {X 0,Y 288.625,Z 541.367,A -85,B 0,C 180,E1 -18483.536,E2 -18483.536} C_VEL
LIN {X 0,Y 291.327,Z 526.523,A -85,B 0,C 180,E1 -18484.419,E2 -18484.419} C_VEL
LIN {X 0,Y 296.562,Z 496.949,A -85,B 0,C 180,E1 -18485.804,E2 -18485.804} C_VEL
LIN {X 0,Y 306.88,Z 443.044,A -85,B 0,C 180,E1 -18488.197,E2 -18488.197} C_VEL
LIN {X 0,Y 304.95,Z 440.484,A -85,B 0,C 180,E1 -18490.19,E2 -18490.19} C_VEL
LIN {X 0,Y 303.951,Z 439.33,A -85,B 0,C 180,E1 -18491.627,E2 -18491.627} C_VEL
LIN {X 0,Y 302.715,Z 439.484,A -85,B 0,C 180,E1 -18494.664,E2 -18494.664} C_VEL
LIN {X 0,Y 302.758,Z 441.296,A -85,B 0,C 180,E1 -18496.967,E2 -18496.967} C_VEL
LIN {X 0,Y 303.495,Z 444.542,A -85,B 0,C 180,E1 -18499.17,E2 -18499.17} C_VEL
LIN {X 0,Y 304.693,Z 449.525,A -85,B 0,C 180,E1 -18501.222,E2 -18501.222} C_VEL
LIN {X 0,Y 305.031,Z 451.863,A -85,B 0,C 180,E1 -18501.849,E2 -18501.849} C_VEL
LIN {X 0,Y 304.729,Z 463.214,A -85,B 0,C 180,E1 -18503.369,E2 -18503.369} C_VEL
LIN {X 0,Y 304.389,Z 471.916,A -85,B 0,C 180,E1 -18504.333,E2 -18504.333} C_VEL
LIN {X 0,Y 293.493,Z 535.928,A -85,B 0,C 180,E1 -18507.195,E2 -18507.195} C_VEL
LIN {X 0,Y 290.486,Z 549.291,A -85,B 0,C 180,E1 -18508.046,E2 -18508.046} C_VEL
LIN {X 0,Y 287.108,Z 561.616,A -85,B 0,C 180,E1 -18509.066,E2 -18509.066} C_VEL
LIN {X 0,Y 283.576,Z 572.91,A -85,B 0,C 180,E1 -18510.286,E2 -18510.286} C_VEL
LIN {X 0,Y 279.818,Z 583.491,A -85,B 0,C 180,E1 -18511.701,E2 -18511.701} C_VEL
LIN {X 0,Y 275.59,Z 594.122,A -85,B 0,C 180,E1 -18513.495,E2 -18513.495} C_VEL
LIN {X 0,Y 271.44,Z 603.665,A -85,B 0,C 180,E1 -18515.527,E2 -18515.527} C_VEL
LIN {X 0,Y 267.684,Z 611.507,A -85,B 0,C 180,E1 -18517.623,E2 -18517.623} C_VEL
LIN {X 0,Y 264.393,Z 617.946,A -85,B 0,C 180,E1 -18519.784,E2 -18519.784} C_VEL
LIN {X 0,Y 261.642,Z 623.135,A -85,B 0,C 180,E1 -18522.007,E2 -18522.007} C_VEL
LIN {X 0,Y 259.463,Z 627.199,A -85,B 0,C 180,E1 -18524.284,E2 -18524.284} C_VEL
LIN {X 0,Y 258.112,Z 629.379,A -85,B 0,C 180,E1 -18525.815,E2 -18525.815} C_VEL
LIN {X 0,Y 256.03,Z 632.405,A -85,B 0,C 180,E1 -18528.922,E2 -18528.922} C_VEL
LIN {X 0,Y 255.286,Z 633.323,A -85,B 0,C 180,E1 -18530.492,E2 -18530.492} C_VEL
LIN {X 0,Y 254.74,Z 633.807,A -85,B 0,C 180,E1 -18532.071,E2 -18532.071} C_VEL
LIN {X 0,Y 254.177,Z 633.76,A -85,B 0,C 180,E1 -18534.518,E2 -18534.518} C_VEL
LIN {X 0,Y 254.014,Z 632.803,A -85,B 0,C 180,E1 -18536.828,E2 -18536.828} C_VEL
LIN {X 0,Y 254.022,Z 631.61,A -85,B 0,C 180,E1 -18538.415,E2 -18538.415} C_VEL
LIN {X 0,Y 253.988,Z 628.985,A -85,B 0,C 180,E1 -18540.793,E2 -18540.793} C_VEL
LIN {X 0,Y 254.172,Z 625.281,A -85,B 0,C 180,E1 -18543.17,E2 -18543.17} C_VEL
LIN {X 0,Y 254.301,Z 619.832,A -85,B 0,C 180,E1 -18545.765,E2 -18545.765} C_VEL
LIN {X 0,Y 254.645,Z 612.854,A -85,B 0,C 180,E1 -18548.331,E2 -18548.331} C_VEL
LIN {X 0,Y 255.129,Z 604.613,A -85,B 0,C 180,E1 -18550.716,E2 -18550.716} C_VEL
LIN {X 0,Y 255.756,Z 596.225,A -85,B 0,C 180,E1 -18552.699,E2 -18552.699} C_VEL
LIN {X 0,Y 256.625,Z 585.991,A -85,B 0,C 180,E1 -18554.674,E2 -18554.674} C_VEL
LIN {X 0,Y 257.612,Z 574.708,A -85,B 0,C 180,E1 -18556.442,E2 -18556.442} C_VEL
LIN {X 0,Y 258.524,Z 562.893,A -85,B 0,C 180,E1 -18557.917,E2 -18557.917} C_VEL
LIN {X 0,Y 259.431,Z 550.066,A -85,B 0,C 180,E1 -18559.176,E2 -18559.176} C_VEL
LIN {X 0,Y 260.305,Z 536.045,A -85,B 0,C 180,E1 -18560.187,E2 -18560.187} C_VEL
LIN {X 0,Y 260.885,Z 522.487,A -85,B 0,C 180,E1 -18560.861,E2 -18560.861} C_VEL
LIN {X 0,Y 263.567,Z 455.178,A -85,B 0,C 180,E1 -18563.753,E2 -18563.753} C_VEL
LIN {X 0,Y 261,Z 427.612,A -85,B 0,C 180,E1 -18565.075,E2 -18565.075} C_VEL
LIN {X 0,Y 260.667,Z 419.93,A -85,B 0,C 180,E1 -18565.462,E2 -18565.462} C_VEL
LIN {X 0,Y 262.748,Z 399.922,A -85,B 0,C 180,E1 -18569.659,E2 -18569.659} C_VEL
LIN {X 0,Y 262.749,Z 396.851,A -85,B 0,C 180,E1 -18570.323,E2 -18570.323} C_VEL
LIN {X 0,Y 258.941,Z 379.517,A -85,B 0,C 180,E1 -18574.383,E2 -18574.383} C_VEL
LIN {X 0,Y 256.206,Z 367.437,A -85,B 0,C 180,E1 -18577.344,E2 -18577.344} C_VEL
LIN {X 0,Y 256.06,Z 367.213,A -85,B 0,C 180,E1 -18581.203,E2 -18581.203} C_VEL
LIN {X 0,Y 256.047,Z 367.181,A -85,B 0,C 180,E1 -18585.533,E2 -18585.533} C_VEL
LIN {X 0,Y 256.093,Z 367.297,A -85,B 0,C 180,E1 -18587.814,E2 -18587.814} C_VEL
LIN {X 0,Y 257.52,Z 372.121,A -85,B 0,C 180,E1 -18590.039,E2 -18590.039} C_VEL
LIN {X 0,Y 260.092,Z 376.708,A -85,B 0,C 180,E1 -18590.752,E2 -18590.752} C_VEL
LIN {X 0,Y 267.93,Z 391.173,A -85,B 0,C 180,E1 -18592.589,E2 -18592.589} C_VEL
LIN {X 0,Y 275.962,Z 407.856,A -85,B 0,C 180,E1 -18594.38,E2 -18594.38} C_VEL
LIN {X 0,Y 281.896,Z 422.166,A -85,B 0,C 180,E1 -18595.674,E2 -18595.674} C_VEL
LIN {X 0,Y 279.294,Z 491.606,A -85,B 0,C 180,E1 -18597.41,E2 -18597.41} C_VEL
LIN {X 0,Y 278.328,Z 511.895,A -85,B 0,C 180,E1 -18597.975,E2 -18597.975} C_VEL
LIN {X 0,Y 276.891,Z 526.485,A -85,B 0,C 180,E1 -18598.644,E2 -18598.644} C_VEL
LIN {X 0,Y 275.207,Z 539.263,A -85,B 0,C 180,E1 -18599.497,E2 -18599.497} C_VEL
LIN {X 0,Y 273.014,Z 552.853,A -85,B 0,C 180,E1 -18600.717,E2 -18600.717} C_VEL
